// TIA Portal V19 export
FUNCTION "ALARM" : Void   // FC6, LAD
{ S7_Optimized_Access := 'TRUE' }
// stored: SetENOAutomatically false
   VAR_TEMP   // added for the SCL form of the ladder/FBD networks
      _w1 : Bool;
      _w2 : Bool;
   END_VAR
BEGIN

REGION Network 1: ALARM RESET (MASTER TO SLAVE)
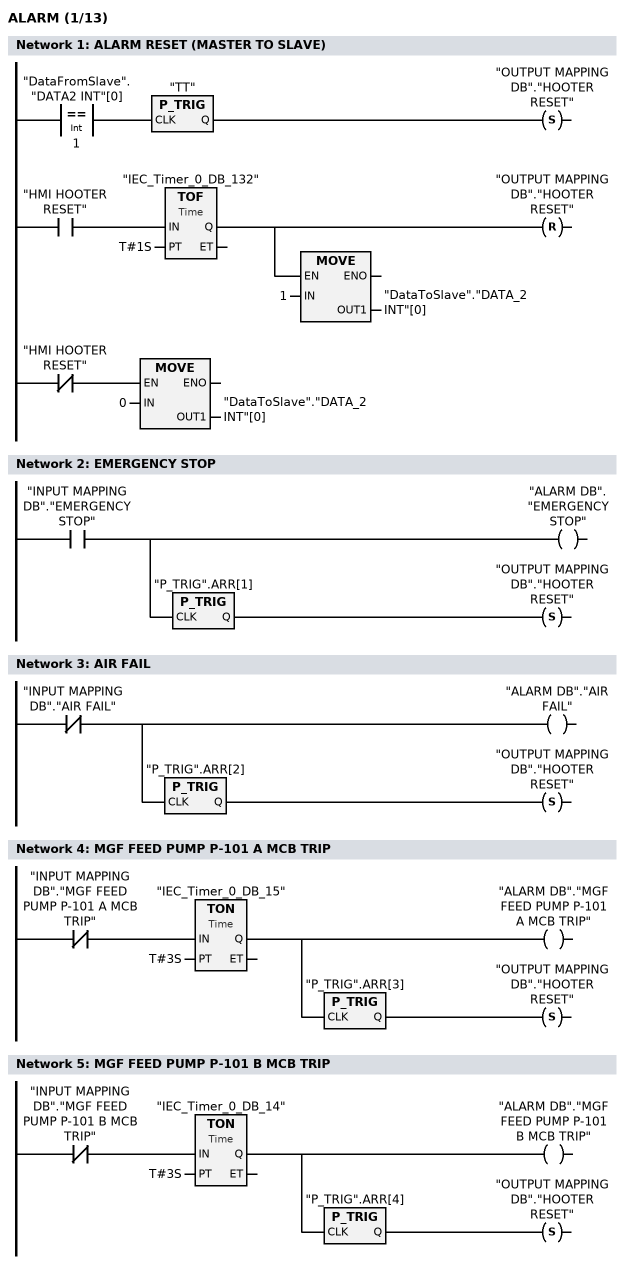
   RUNG wire#powerrail
      { S7_Templates := "SrcType := Int" } EQ_Contact(in1 := "DataFromSlave"."DATA2 INT"[0], in2 := 1)
      P_Trig( "TT" )
      S_Coil( "OUTPUT MAPPING DB"."HOOTER RESET" )
   END_RUNG
   RUNG wire#powerrail
      Contact( "HMI HOOTER RESET" )
      { S7_Templates := "time_type := Time" } "IEC_Timer_0_DB_132".TOF(pt := T#1S, et =>)
      wire#w1
      R_Coil( "OUTPUT MAPPING DB"."HOOTER RESET" )
   END_RUNG
   RUNG wire#w1
      Move(in := 1, out1 => "DataToSlave"."DATA_2 INT"[0])
   END_RUNG
   RUNG wire#powerrail
      I_Contact( "HMI HOOTER RESET" )
      Move(in := 0, out1 => "DataToSlave"."DATA_2 INT"[0])
   END_RUNG
   // the same network as SCL:
   #_w1 := "DataFromSlave"."DATA2 INT"[0] = 1;
   #_w2 := #_w1 AND NOT "TT";   // rising edge
   "TT" := #_w1;
   IF #_w2 THEN "OUTPUT MAPPING DB"."HOOTER RESET" := TRUE; END_IF;
   "IEC_Timer_0_DB_132".TOF(IN := "HMI HOOTER RESET", PT := T#1S);
   IF "IEC_Timer_0_DB_132".Q THEN
       "OUTPUT MAPPING DB"."HOOTER RESET" := FALSE;
       "DataToSlave"."DATA_2 INT"[0] := 1;
   END_IF;
   IF NOT "HMI HOOTER RESET" THEN "DataToSlave"."DATA_2 INT"[0] := 0; END_IF;
END_REGION

REGION Network 2: EMERGENCY STOP
   RUNG wire#powerrail
      Contact( "INPUT MAPPING DB"."EMERGENCY STOP" )
      wire#w1
      Coil( "ALARM DB"."EMERGENCY STOP" )
   END_RUNG
   RUNG wire#w1
      P_Trig( "P_TRIG".ARR[1] )
      S_Coil( "OUTPUT MAPPING DB"."HOOTER RESET" )
   END_RUNG
   // the same network as SCL:
   "ALARM DB"."EMERGENCY STOP" := "INPUT MAPPING DB"."EMERGENCY STOP";
   #_w1 := "INPUT MAPPING DB"."EMERGENCY STOP" AND NOT "P_TRIG".ARR[1];   // rising edge
   "P_TRIG".ARR[1] := "INPUT MAPPING DB"."EMERGENCY STOP";
   IF #_w1 THEN "OUTPUT MAPPING DB"."HOOTER RESET" := TRUE; END_IF;
END_REGION

REGION Network 3: AIR FAIL
   RUNG wire#powerrail
      I_Contact( "INPUT MAPPING DB"."AIR FAIL" )
      wire#w1
      Coil( "ALARM DB"."AIR FAIL" )
   END_RUNG
   RUNG wire#w1
      P_Trig( "P_TRIG".ARR[2] )
      S_Coil( "OUTPUT MAPPING DB"."HOOTER RESET" )
   END_RUNG
   // the same network as SCL:
   "ALARM DB"."AIR FAIL" := NOT "INPUT MAPPING DB"."AIR FAIL";
   #_w1 := NOT "INPUT MAPPING DB"."AIR FAIL" AND NOT "P_TRIG".ARR[2];   // rising edge
   "P_TRIG".ARR[2] := NOT "INPUT MAPPING DB"."AIR FAIL";
   IF #_w1 THEN "OUTPUT MAPPING DB"."HOOTER RESET" := TRUE; END_IF;
END_REGION

REGION Network 4: MGF FEED PUMP P-101 A MCB TRIP
   RUNG wire#powerrail
      I_Contact( "INPUT MAPPING DB"."MGF FEED PUMP P-101 A MCB TRIP" )
      { S7_Templates := "time_type := Time" } "IEC_Timer_0_DB_15".TON(pt := T#3S, et =>)
      wire#w1
      Coil( "ALARM DB"."MGF FEED PUMP P-101 A MCB TRIP" )
   END_RUNG
   RUNG wire#w1
      P_Trig( "P_TRIG".ARR[3] )
      S_Coil( "OUTPUT MAPPING DB"."HOOTER RESET" )
   END_RUNG
   // the same network as SCL:
   "IEC_Timer_0_DB_15".TON(IN := NOT "INPUT MAPPING DB"."MGF FEED PUMP P-101 A MCB TRIP", PT := T#3S);
   "ALARM DB"."MGF FEED PUMP P-101 A MCB TRIP" := "IEC_Timer_0_DB_15".Q;
   #_w1 := "IEC_Timer_0_DB_15".Q AND NOT "P_TRIG".ARR[3];   // rising edge
   "P_TRIG".ARR[3] := "IEC_Timer_0_DB_15".Q;
   IF #_w1 THEN "OUTPUT MAPPING DB"."HOOTER RESET" := TRUE; END_IF;
END_REGION

REGION Network 5: MGF FEED PUMP P-101 B MCB TRIP
   RUNG wire#powerrail
      I_Contact( "INPUT MAPPING DB"."MGF FEED PUMP P-101 B MCB TRIP" )
      { S7_Templates := "time_type := Time" } "IEC_Timer_0_DB_14".TON(pt := T#3S, et =>)
      wire#w1
      Coil( "ALARM DB"."MGF FEED PUMP P-101 B MCB TRIP" )
   END_RUNG
   RUNG wire#w1
      P_Trig( "P_TRIG".ARR[4] )
      S_Coil( "OUTPUT MAPPING DB"."HOOTER RESET" )
   END_RUNG
   // the same network as SCL:
   "IEC_Timer_0_DB_14".TON(IN := NOT "INPUT MAPPING DB"."MGF FEED PUMP P-101 B MCB TRIP", PT := T#3S);
   "ALARM DB"."MGF FEED PUMP P-101 B MCB TRIP" := "IEC_Timer_0_DB_14".Q;
   #_w1 := "IEC_Timer_0_DB_14".Q AND NOT "P_TRIG".ARR[4];   // rising edge
   "P_TRIG".ARR[4] := "IEC_Timer_0_DB_14".Q;
   IF #_w1 THEN "OUTPUT MAPPING DB"."HOOTER RESET" := TRUE; END_IF;
END_REGION

REGION Network 6: MGF BACK WASH P-102 A MCB TRIP
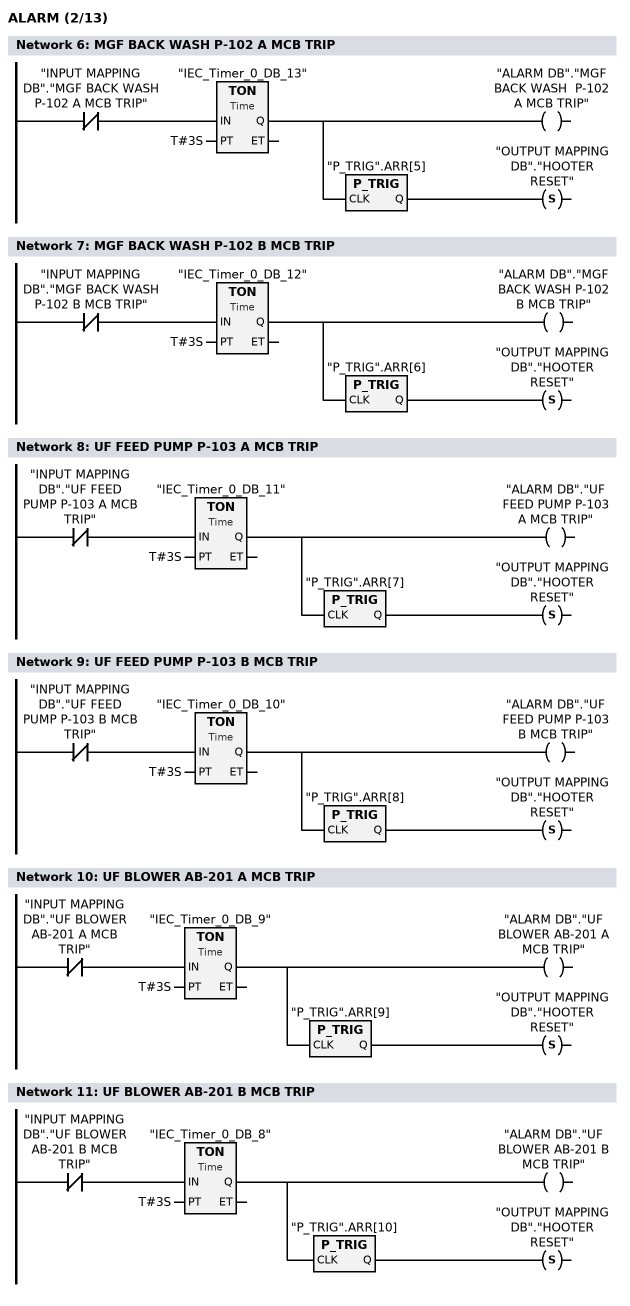
   RUNG wire#powerrail
      I_Contact( "INPUT MAPPING DB"."MGF BACK WASH  P-102 A MCB TRIP" )
      { S7_Templates := "time_type := Time" } "IEC_Timer_0_DB_13".TON(pt := T#3S, et =>)
      wire#w1
      Coil( "ALARM DB"."MGF BACK WASH  P-102 A MCB TRIP" )
   END_RUNG
   RUNG wire#w1
      P_Trig( "P_TRIG".ARR[5] )
      S_Coil( "OUTPUT MAPPING DB"."HOOTER RESET" )
   END_RUNG
   // the same network as SCL:
   "IEC_Timer_0_DB_13".TON(IN := NOT "INPUT MAPPING DB"."MGF BACK WASH  P-102 A MCB TRIP", PT := T#3S);
   "ALARM DB"."MGF BACK WASH  P-102 A MCB TRIP" := "IEC_Timer_0_DB_13".Q;
   #_w1 := "IEC_Timer_0_DB_13".Q AND NOT "P_TRIG".ARR[5];   // rising edge
   "P_TRIG".ARR[5] := "IEC_Timer_0_DB_13".Q;
   IF #_w1 THEN "OUTPUT MAPPING DB"."HOOTER RESET" := TRUE; END_IF;
END_REGION

REGION Network 7: MGF BACK WASH P-102 B MCB TRIP
   RUNG wire#powerrail
      I_Contact( "INPUT MAPPING DB"."MGF BACK WASH P-102 B MCB TRIP" )
      { S7_Templates := "time_type := Time" } "IEC_Timer_0_DB_12".TON(pt := T#3S, et =>)
      wire#w1
      Coil( "ALARM DB"."MGF BACK WASH P-102 B MCB TRIP" )
   END_RUNG
   RUNG wire#w1
      P_Trig( "P_TRIG".ARR[6] )
      S_Coil( "OUTPUT MAPPING DB"."HOOTER RESET" )
   END_RUNG
   // the same network as SCL:
   "IEC_Timer_0_DB_12".TON(IN := NOT "INPUT MAPPING DB"."MGF BACK WASH P-102 B MCB TRIP", PT := T#3S);
   "ALARM DB"."MGF BACK WASH P-102 B MCB TRIP" := "IEC_Timer_0_DB_12".Q;
   #_w1 := "IEC_Timer_0_DB_12".Q AND NOT "P_TRIG".ARR[6];   // rising edge
   "P_TRIG".ARR[6] := "IEC_Timer_0_DB_12".Q;
   IF #_w1 THEN "OUTPUT MAPPING DB"."HOOTER RESET" := TRUE; END_IF;
END_REGION

REGION Network 8: UF FEED PUMP P-103 A MCB TRIP
   RUNG wire#powerrail
      I_Contact( "INPUT MAPPING DB"."UF FEED PUMP P-103 A MCB TRIP" )
      { S7_Templates := "time_type := Time" } "IEC_Timer_0_DB_11".TON(pt := T#3S, et =>)
      wire#w1
      Coil( "ALARM DB"."UF FEED PUMP P-103 A MCB TRIP" )
   END_RUNG
   RUNG wire#w1
      P_Trig( "P_TRIG".ARR[7] )
      S_Coil( "OUTPUT MAPPING DB"."HOOTER RESET" )
   END_RUNG
   // the same network as SCL:
   "IEC_Timer_0_DB_11".TON(IN := NOT "INPUT MAPPING DB"."UF FEED PUMP P-103 A MCB TRIP", PT := T#3S);
   "ALARM DB"."UF FEED PUMP P-103 A MCB TRIP" := "IEC_Timer_0_DB_11".Q;
   #_w1 := "IEC_Timer_0_DB_11".Q AND NOT "P_TRIG".ARR[7];   // rising edge
   "P_TRIG".ARR[7] := "IEC_Timer_0_DB_11".Q;
   IF #_w1 THEN "OUTPUT MAPPING DB"."HOOTER RESET" := TRUE; END_IF;
END_REGION

REGION Network 9: UF FEED PUMP P-103 B MCB TRIP
   RUNG wire#powerrail
      I_Contact( "INPUT MAPPING DB"."UF FEED PUMP P-103 B MCB TRIP" )
      { S7_Templates := "time_type := Time" } "IEC_Timer_0_DB_10".TON(pt := T#3S, et =>)
      wire#w1
      Coil( "ALARM DB"."UF FEED PUMP P-103 B MCB TRIP" )
   END_RUNG
   RUNG wire#w1
      P_Trig( "P_TRIG".ARR[8] )
      S_Coil( "OUTPUT MAPPING DB"."HOOTER RESET" )
   END_RUNG
   // the same network as SCL:
   "IEC_Timer_0_DB_10".TON(IN := NOT "INPUT MAPPING DB"."UF FEED PUMP P-103 B MCB TRIP", PT := T#3S);
   "ALARM DB"."UF FEED PUMP P-103 B MCB TRIP" := "IEC_Timer_0_DB_10".Q;
   #_w1 := "IEC_Timer_0_DB_10".Q AND NOT "P_TRIG".ARR[8];   // rising edge
   "P_TRIG".ARR[8] := "IEC_Timer_0_DB_10".Q;
   IF #_w1 THEN "OUTPUT MAPPING DB"."HOOTER RESET" := TRUE; END_IF;
END_REGION

REGION Network 10: UF BLOWER AB-201 A MCB TRIP
   RUNG wire#powerrail
      I_Contact( "INPUT MAPPING DB"."UF BLOWER AB-201 A MCB TRIP" )
      { S7_Templates := "time_type := Time" } "IEC_Timer_0_DB_9".TON(pt := T#3S, et =>)
      wire#w1
      Coil( "ALARM DB"."UF BLOWER AB-201 A MCB TRIP" )
   END_RUNG
   RUNG wire#w1
      P_Trig( "P_TRIG".ARR[9] )
      S_Coil( "OUTPUT MAPPING DB"."HOOTER RESET" )
   END_RUNG
   // the same network as SCL:
   "IEC_Timer_0_DB_9".TON(IN := NOT "INPUT MAPPING DB"."UF BLOWER AB-201 A MCB TRIP", PT := T#3S);
   "ALARM DB"."UF BLOWER AB-201 A MCB TRIP" := "IEC_Timer_0_DB_9".Q;
   #_w1 := "IEC_Timer_0_DB_9".Q AND NOT "P_TRIG".ARR[9];   // rising edge
   "P_TRIG".ARR[9] := "IEC_Timer_0_DB_9".Q;
   IF #_w1 THEN "OUTPUT MAPPING DB"."HOOTER RESET" := TRUE; END_IF;
END_REGION

REGION Network 11: UF BLOWER AB-201 B MCB TRIP
   RUNG wire#powerrail
      I_Contact( "INPUT MAPPING DB"."UF BLOWER AB-201 B MCB TRIP" )
      { S7_Templates := "time_type := Time" } "IEC_Timer_0_DB_8".TON(pt := T#3S, et =>)
      wire#w1
      Coil( "ALARM DB"."UF BLOWER AB-201 B MCB TRIP" )
   END_RUNG
   RUNG wire#w1
      P_Trig( "P_TRIG".ARR[10] )
      S_Coil( "OUTPUT MAPPING DB"."HOOTER RESET" )
   END_RUNG
   // the same network as SCL:
   "IEC_Timer_0_DB_8".TON(IN := NOT "INPUT MAPPING DB"."UF BLOWER AB-201 B MCB TRIP", PT := T#3S);
   "ALARM DB"."UF BLOWER AB-201 B MCB TRIP" := "IEC_Timer_0_DB_8".Q;
   #_w1 := "IEC_Timer_0_DB_8".Q AND NOT "P_TRIG".ARR[10];   // rising edge
   "P_TRIG".ARR[10] := "IEC_Timer_0_DB_8".Q;
   IF #_w1 THEN "OUTPUT MAPPING DB"."HOOTER RESET" := TRUE; END_IF;
END_REGION

REGION Network 12: DM FEED PUMP P-502 A MPCB TRIP
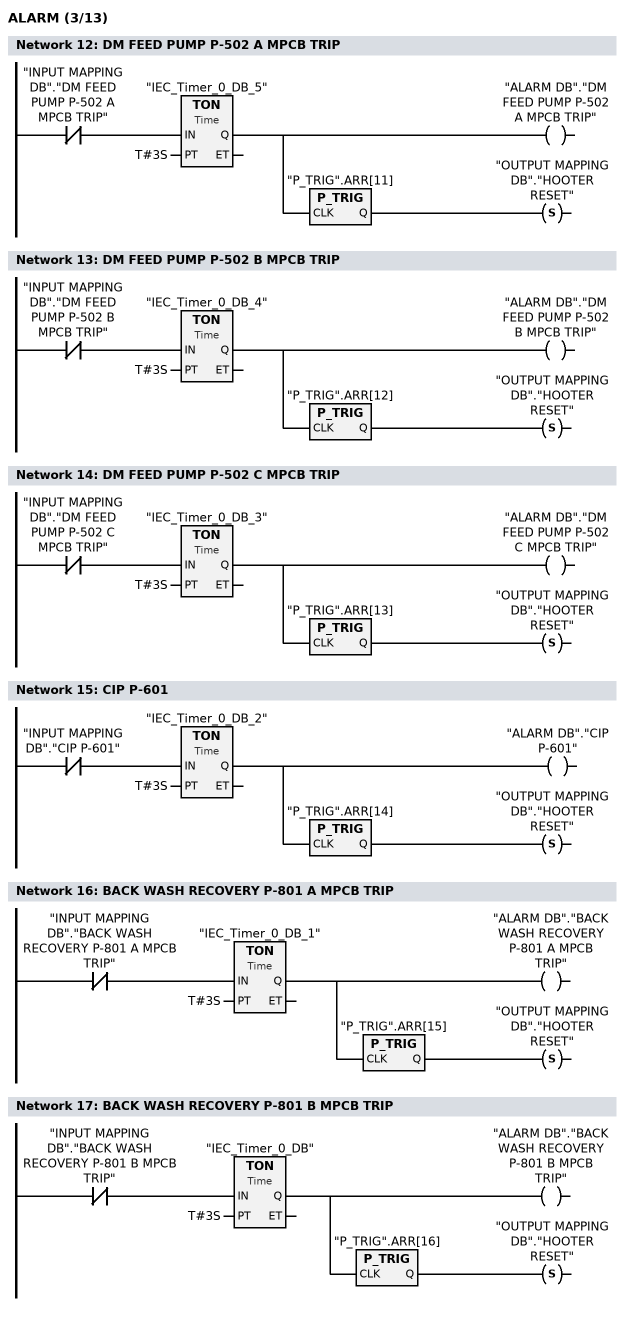
   RUNG wire#powerrail
      I_Contact( "INPUT MAPPING DB"."DM FEED PUMP P-502 A MPCB TRIP" )
      { S7_Templates := "time_type := Time" } "IEC_Timer_0_DB_5".TON(pt := T#3S, et =>)
      wire#w1
      Coil( "ALARM DB"."DM FEED PUMP P-502 A MPCB TRIP" )
   END_RUNG
   RUNG wire#w1
      P_Trig( "P_TRIG".ARR[11] )
      S_Coil( "OUTPUT MAPPING DB"."HOOTER RESET" )
   END_RUNG
   // the same network as SCL:
   "IEC_Timer_0_DB_5".TON(IN := NOT "INPUT MAPPING DB"."DM FEED PUMP P-502 A MPCB TRIP", PT := T#3S);
   "ALARM DB"."DM FEED PUMP P-502 A MPCB TRIP" := "IEC_Timer_0_DB_5".Q;
   #_w1 := "IEC_Timer_0_DB_5".Q AND NOT "P_TRIG".ARR[11];   // rising edge
   "P_TRIG".ARR[11] := "IEC_Timer_0_DB_5".Q;
   IF #_w1 THEN "OUTPUT MAPPING DB"."HOOTER RESET" := TRUE; END_IF;
END_REGION

REGION Network 13: DM FEED PUMP P-502 B MPCB TRIP
   RUNG wire#powerrail
      I_Contact( "INPUT MAPPING DB"."DM FEED PUMP P-502 B MPCB TRIP" )
      { S7_Templates := "time_type := Time" } "IEC_Timer_0_DB_4".TON(pt := T#3S, et =>)
      wire#w1
      Coil( "ALARM DB"."DM FEED PUMP P-502 B MPCB TRIP" )
   END_RUNG
   RUNG wire#w1
      P_Trig( "P_TRIG".ARR[12] )
      S_Coil( "OUTPUT MAPPING DB"."HOOTER RESET" )
   END_RUNG
   // the same network as SCL:
   "IEC_Timer_0_DB_4".TON(IN := NOT "INPUT MAPPING DB"."DM FEED PUMP P-502 B MPCB TRIP", PT := T#3S);
   "ALARM DB"."DM FEED PUMP P-502 B MPCB TRIP" := "IEC_Timer_0_DB_4".Q;
   #_w1 := "IEC_Timer_0_DB_4".Q AND NOT "P_TRIG".ARR[12];   // rising edge
   "P_TRIG".ARR[12] := "IEC_Timer_0_DB_4".Q;
   IF #_w1 THEN "OUTPUT MAPPING DB"."HOOTER RESET" := TRUE; END_IF;
END_REGION

REGION Network 14: DM FEED PUMP P-502 C MPCB TRIP
   RUNG wire#powerrail
      I_Contact( "INPUT MAPPING DB"."DM FEED PUMP P-502 C MPCB TRIP" )
      { S7_Templates := "time_type := Time" } "IEC_Timer_0_DB_3".TON(pt := T#3S, et =>)
      wire#w1
      Coil( "ALARM DB"."DM FEED PUMP P-502 C MPCB TRIP" )
   END_RUNG
   RUNG wire#w1
      P_Trig( "P_TRIG".ARR[13] )
      S_Coil( "OUTPUT MAPPING DB"."HOOTER RESET" )
   END_RUNG
   // the same network as SCL:
   "IEC_Timer_0_DB_3".TON(IN := NOT "INPUT MAPPING DB"."DM FEED PUMP P-502 C MPCB TRIP", PT := T#3S);
   "ALARM DB"."DM FEED PUMP P-502 C MPCB TRIP" := "IEC_Timer_0_DB_3".Q;
   #_w1 := "IEC_Timer_0_DB_3".Q AND NOT "P_TRIG".ARR[13];   // rising edge
   "P_TRIG".ARR[13] := "IEC_Timer_0_DB_3".Q;
   IF #_w1 THEN "OUTPUT MAPPING DB"."HOOTER RESET" := TRUE; END_IF;
END_REGION

REGION Network 15: CIP P-601
   RUNG wire#powerrail
      I_Contact( "INPUT MAPPING DB"."CIP P-601" )
      { S7_Templates := "time_type := Time" } "IEC_Timer_0_DB_2".TON(pt := T#3S, et =>)
      wire#w1
      Coil( "ALARM DB"."CIP P-601" )
   END_RUNG
   RUNG wire#w1
      P_Trig( "P_TRIG".ARR[14] )
      S_Coil( "OUTPUT MAPPING DB"."HOOTER RESET" )
   END_RUNG
   // the same network as SCL:
   "IEC_Timer_0_DB_2".TON(IN := NOT "INPUT MAPPING DB"."CIP P-601", PT := T#3S);
   "ALARM DB"."CIP P-601" := "IEC_Timer_0_DB_2".Q;
   #_w1 := "IEC_Timer_0_DB_2".Q AND NOT "P_TRIG".ARR[14];   // rising edge
   "P_TRIG".ARR[14] := "IEC_Timer_0_DB_2".Q;
   IF #_w1 THEN "OUTPUT MAPPING DB"."HOOTER RESET" := TRUE; END_IF;
END_REGION

REGION Network 16: BACK WASH RECOVERY P-801 A MPCB TRIP
   RUNG wire#powerrail
      I_Contact( "INPUT MAPPING DB"."BACK WASH RECOVERY P-801 A MPCB TRIP" )
      { S7_Templates := "time_type := Time" } "IEC_Timer_0_DB_1".TON(pt := T#3S, et =>)
      wire#w1
      Coil( "ALARM DB"."BACK WASH RECOVERY P-801 A MPCB TRIP" )
   END_RUNG
   RUNG wire#w1
      P_Trig( "P_TRIG".ARR[15] )
      S_Coil( "OUTPUT MAPPING DB"."HOOTER RESET" )
   END_RUNG
   // the same network as SCL:
   "IEC_Timer_0_DB_1".TON(IN := NOT "INPUT MAPPING DB"."BACK WASH RECOVERY P-801 A MPCB TRIP", PT := T#3S);
   "ALARM DB"."BACK WASH RECOVERY P-801 A MPCB TRIP" := "IEC_Timer_0_DB_1".Q;
   #_w1 := "IEC_Timer_0_DB_1".Q AND NOT "P_TRIG".ARR[15];   // rising edge
   "P_TRIG".ARR[15] := "IEC_Timer_0_DB_1".Q;
   IF #_w1 THEN "OUTPUT MAPPING DB"."HOOTER RESET" := TRUE; END_IF;
END_REGION

REGION Network 17: BACK WASH RECOVERY P-801 B MPCB TRIP
   RUNG wire#powerrail
      I_Contact( "INPUT MAPPING DB"."BACK WASH RECOVERY P-801 B MPCB TRIP" )
      { S7_Templates := "time_type := Time" } "IEC_Timer_0_DB".TON(pt := T#3S, et =>)
      wire#w1
      Coil( "ALARM DB"."BACK WASH RECOVERY P-801 B MPCB TRIP" )
   END_RUNG
   RUNG wire#w1
      P_Trig( "P_TRIG".ARR[16] )
      S_Coil( "OUTPUT MAPPING DB"."HOOTER RESET" )
   END_RUNG
   // the same network as SCL:
   "IEC_Timer_0_DB".TON(IN := NOT "INPUT MAPPING DB"."BACK WASH RECOVERY P-801 B MPCB TRIP", PT := T#3S);
   "ALARM DB"."BACK WASH RECOVERY P-801 B MPCB TRIP" := "IEC_Timer_0_DB".Q;
   #_w1 := "IEC_Timer_0_DB".Q AND NOT "P_TRIG".ARR[16];   // rising edge
   "P_TRIG".ARR[16] := "IEC_Timer_0_DB".Q;
   IF #_w1 THEN "OUTPUT MAPPING DB"."HOOTER RESET" := TRUE; END_IF;
END_REGION

REGION Network 18: UF BACKWASH P-201A TRIP
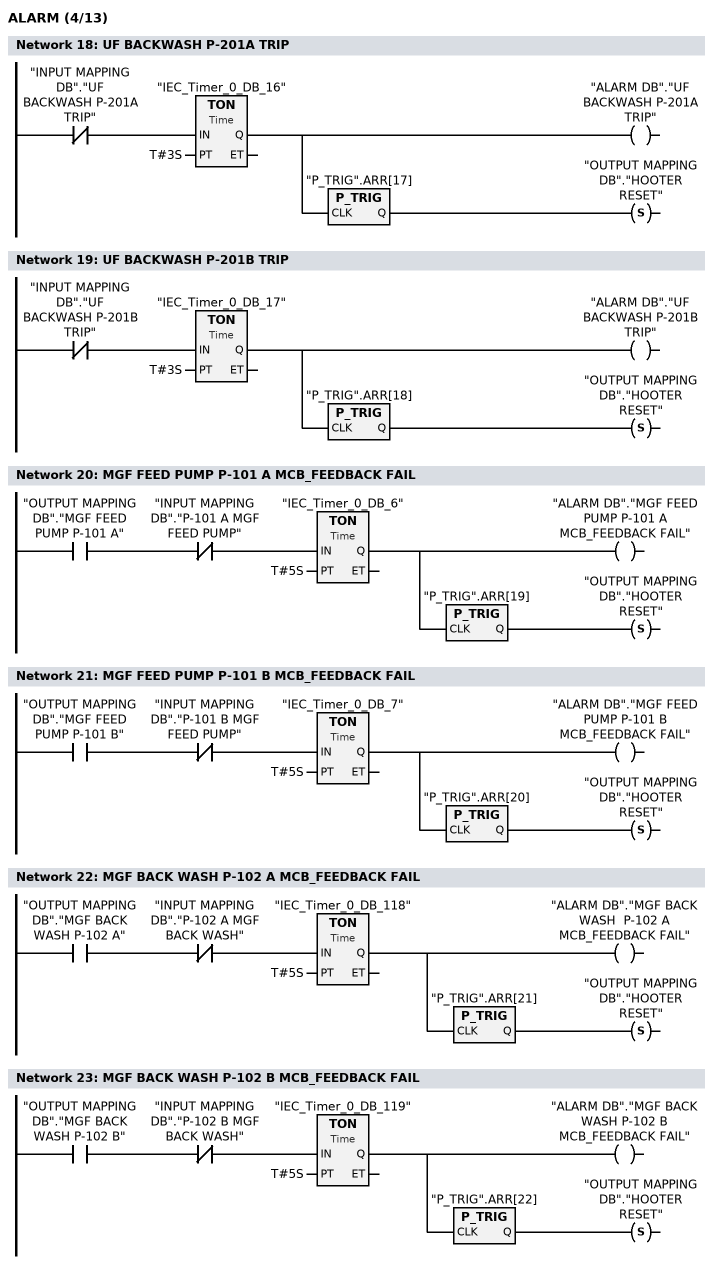
   RUNG wire#powerrail
      I_Contact( "INPUT MAPPING DB"."UF BACKWASH P-201A TRIP" )
      { S7_Templates := "time_type := Time" } "IEC_Timer_0_DB_16".TON(pt := T#3S, et =>)
      wire#w1
      Coil( "ALARM DB"."UF BACKWASH P-201A TRIP" )
   END_RUNG
   RUNG wire#w1
      P_Trig( "P_TRIG".ARR[17] )
      S_Coil( "OUTPUT MAPPING DB"."HOOTER RESET" )
   END_RUNG
   // the same network as SCL:
   "IEC_Timer_0_DB_16".TON(IN := NOT "INPUT MAPPING DB"."UF BACKWASH P-201A TRIP", PT := T#3S);
   "ALARM DB"."UF BACKWASH P-201A TRIP" := "IEC_Timer_0_DB_16".Q;
   #_w1 := "IEC_Timer_0_DB_16".Q AND NOT "P_TRIG".ARR[17];   // rising edge
   "P_TRIG".ARR[17] := "IEC_Timer_0_DB_16".Q;
   IF #_w1 THEN "OUTPUT MAPPING DB"."HOOTER RESET" := TRUE; END_IF;
END_REGION

REGION Network 19: UF BACKWASH P-201B TRIP
   RUNG wire#powerrail
      I_Contact( "INPUT MAPPING DB"."UF BACKWASH P-201B TRIP" )
      { S7_Templates := "time_type := Time" } "IEC_Timer_0_DB_17".TON(pt := T#3S, et =>)
      wire#w1
      Coil( "ALARM DB"."UF BACKWASH P-201B TRIP" )
   END_RUNG
   RUNG wire#w1
      P_Trig( "P_TRIG".ARR[18] )
      S_Coil( "OUTPUT MAPPING DB"."HOOTER RESET" )
   END_RUNG
   // the same network as SCL:
   "IEC_Timer_0_DB_17".TON(IN := NOT "INPUT MAPPING DB"."UF BACKWASH P-201B TRIP", PT := T#3S);
   "ALARM DB"."UF BACKWASH P-201B TRIP" := "IEC_Timer_0_DB_17".Q;
   #_w1 := "IEC_Timer_0_DB_17".Q AND NOT "P_TRIG".ARR[18];   // rising edge
   "P_TRIG".ARR[18] := "IEC_Timer_0_DB_17".Q;
   IF #_w1 THEN "OUTPUT MAPPING DB"."HOOTER RESET" := TRUE; END_IF;
END_REGION

REGION Network 20: MGF FEED PUMP P-101 A MCB_FEEDBACK FAIL
   RUNG wire#powerrail
      Contact( "OUTPUT MAPPING DB"."MGF FEED PUMP P-101 A" )
      I_Contact( "INPUT MAPPING DB"."P-101 A MGF FEED PUMP" )
      { S7_Templates := "time_type := Time" } "IEC_Timer_0_DB_6".TON(pt := T#5S, et =>)
      wire#w1
      Coil( "ALARM DB"."MGF FEED PUMP P-101 A MCB_FEEDBACK FAIL" )
   END_RUNG
   RUNG wire#w1
      P_Trig( "P_TRIG".ARR[19] )
      S_Coil( "OUTPUT MAPPING DB"."HOOTER RESET" )
   END_RUNG
   // the same network as SCL:
   "IEC_Timer_0_DB_6".TON(IN := "OUTPUT MAPPING DB"."MGF FEED PUMP P-101 A" AND NOT "INPUT MAPPING DB"."P-101 A MGF FEED PUMP",
                          PT := T#5S);
   "ALARM DB"."MGF FEED PUMP P-101 A MCB_FEEDBACK FAIL" := "IEC_Timer_0_DB_6".Q;
   #_w1 := "IEC_Timer_0_DB_6".Q AND NOT "P_TRIG".ARR[19];   // rising edge
   "P_TRIG".ARR[19] := "IEC_Timer_0_DB_6".Q;
   IF #_w1 THEN "OUTPUT MAPPING DB"."HOOTER RESET" := TRUE; END_IF;
END_REGION

REGION Network 21: MGF FEED PUMP P-101 B MCB_FEEDBACK FAIL
   RUNG wire#powerrail
      Contact( "OUTPUT MAPPING DB"."MGF FEED PUMP P-101 B" )
      I_Contact( "INPUT MAPPING DB"."P-101 B MGF FEED PUMP" )
      { S7_Templates := "time_type := Time" } "IEC_Timer_0_DB_7".TON(pt := T#5S, et =>)
      wire#w1
      Coil( "ALARM DB"."MGF FEED PUMP P-101 B MCB_FEEDBACK FAIL" )
   END_RUNG
   RUNG wire#w1
      P_Trig( "P_TRIG".ARR[20] )
      S_Coil( "OUTPUT MAPPING DB"."HOOTER RESET" )
   END_RUNG
   // the same network as SCL:
   "IEC_Timer_0_DB_7".TON(IN := "OUTPUT MAPPING DB"."MGF FEED PUMP P-101 B" AND NOT "INPUT MAPPING DB"."P-101 B MGF FEED PUMP",
                          PT := T#5S);
   "ALARM DB"."MGF FEED PUMP P-101 B MCB_FEEDBACK FAIL" := "IEC_Timer_0_DB_7".Q;
   #_w1 := "IEC_Timer_0_DB_7".Q AND NOT "P_TRIG".ARR[20];   // rising edge
   "P_TRIG".ARR[20] := "IEC_Timer_0_DB_7".Q;
   IF #_w1 THEN "OUTPUT MAPPING DB"."HOOTER RESET" := TRUE; END_IF;
END_REGION

REGION Network 22: MGF BACK WASH P-102 A MCB_FEEDBACK FAIL
   RUNG wire#powerrail
      Contact( "OUTPUT MAPPING DB"."MGF BACK WASH P-102 A" )
      I_Contact( "INPUT MAPPING DB"."P-102 A MGF BACK WASH" )
      { S7_Templates := "time_type := Time" } "IEC_Timer_0_DB_118".TON(pt := T#5S, et =>)
      wire#w1
      Coil( "ALARM DB"."MGF BACK WASH  P-102 A MCB_FEEDBACK FAIL" )
   END_RUNG
   RUNG wire#w1
      P_Trig( "P_TRIG".ARR[21] )
      S_Coil( "OUTPUT MAPPING DB"."HOOTER RESET" )
   END_RUNG
   // the same network as SCL:
   "IEC_Timer_0_DB_118".TON(IN := "OUTPUT MAPPING DB"."MGF BACK WASH P-102 A" AND NOT "INPUT MAPPING DB"."P-102 A MGF BACK WASH",
                           PT := T#5S);
   "ALARM DB"."MGF BACK WASH  P-102 A MCB_FEEDBACK FAIL" := "IEC_Timer_0_DB_118".Q;
   #_w1 := "IEC_Timer_0_DB_118".Q AND NOT "P_TRIG".ARR[21];   // rising edge
   "P_TRIG".ARR[21] := "IEC_Timer_0_DB_118".Q;
   IF #_w1 THEN "OUTPUT MAPPING DB"."HOOTER RESET" := TRUE; END_IF;
END_REGION

REGION Network 23: MGF BACK WASH P-102 B MCB_FEEDBACK FAIL
   RUNG wire#powerrail
      Contact( "OUTPUT MAPPING DB"."MGF BACK WASH P-102 B" )
      I_Contact( "INPUT MAPPING DB"."P-102 B MGF BACK WASH" )
      { S7_Templates := "time_type := Time" } "IEC_Timer_0_DB_119".TON(pt := T#5S, et =>)
      wire#w1
      Coil( "ALARM DB"."MGF BACK WASH P-102 B MCB_FEEDBACK FAIL" )
   END_RUNG
   RUNG wire#w1
      P_Trig( "P_TRIG".ARR[22] )
      S_Coil( "OUTPUT MAPPING DB"."HOOTER RESET" )
   END_RUNG
   // the same network as SCL:
   "IEC_Timer_0_DB_119".TON(IN := "OUTPUT MAPPING DB"."MGF BACK WASH P-102 B" AND NOT "INPUT MAPPING DB"."P-102 B MGF BACK WASH",
                           PT := T#5S);
   "ALARM DB"."MGF BACK WASH P-102 B MCB_FEEDBACK FAIL" := "IEC_Timer_0_DB_119".Q;
   #_w1 := "IEC_Timer_0_DB_119".Q AND NOT "P_TRIG".ARR[22];   // rising edge
   "P_TRIG".ARR[22] := "IEC_Timer_0_DB_119".Q;
   IF #_w1 THEN "OUTPUT MAPPING DB"."HOOTER RESET" := TRUE; END_IF;
END_REGION

REGION Network 24: UF FEED PUMP P-103 A MCB_FEEDBACK FAIL
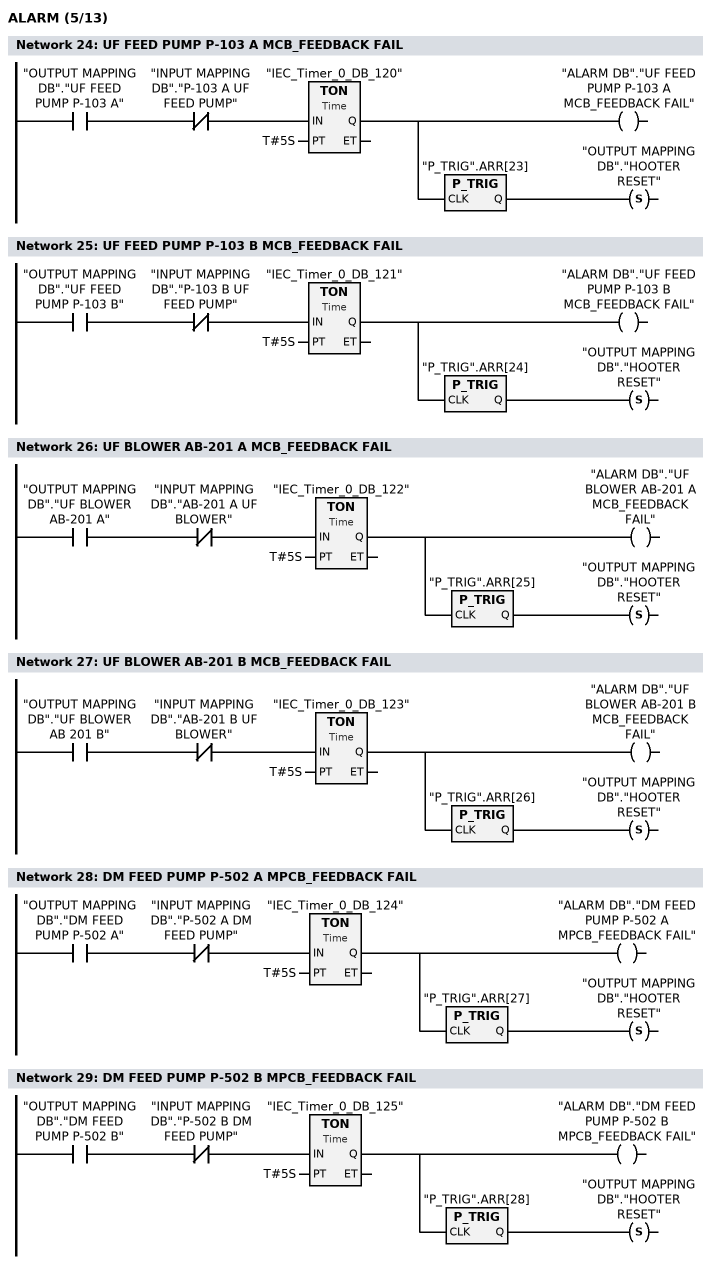
   RUNG wire#powerrail
      Contact( "OUTPUT MAPPING DB"."UF FEED PUMP P-103 A" )
      I_Contact( "INPUT MAPPING DB"."P-103 A UF FEED PUMP" )
      { S7_Templates := "time_type := Time" } "IEC_Timer_0_DB_120".TON(pt := T#5S, et =>)
      wire#w1
      Coil( "ALARM DB"."UF FEED PUMP P-103 A MCB_FEEDBACK FAIL" )
   END_RUNG
   RUNG wire#w1
      P_Trig( "P_TRIG".ARR[23] )
      S_Coil( "OUTPUT MAPPING DB"."HOOTER RESET" )
   END_RUNG
   // the same network as SCL:
   "IEC_Timer_0_DB_120".TON(IN := "OUTPUT MAPPING DB"."UF FEED PUMP P-103 A" AND NOT "INPUT MAPPING DB"."P-103 A UF FEED PUMP",
                           PT := T#5S);
   "ALARM DB"."UF FEED PUMP P-103 A MCB_FEEDBACK FAIL" := "IEC_Timer_0_DB_120".Q;
   #_w1 := "IEC_Timer_0_DB_120".Q AND NOT "P_TRIG".ARR[23];   // rising edge
   "P_TRIG".ARR[23] := "IEC_Timer_0_DB_120".Q;
   IF #_w1 THEN "OUTPUT MAPPING DB"."HOOTER RESET" := TRUE; END_IF;
END_REGION

REGION Network 25: UF FEED PUMP P-103 B MCB_FEEDBACK FAIL
   RUNG wire#powerrail
      Contact( "OUTPUT MAPPING DB"."UF FEED PUMP P-103 B" )
      I_Contact( "INPUT MAPPING DB"."P-103 B UF FEED PUMP" )
      { S7_Templates := "time_type := Time" } "IEC_Timer_0_DB_121".TON(pt := T#5S, et =>)
      wire#w1
      Coil( "ALARM DB"."UF FEED PUMP P-103 B MCB_FEEDBACK FAIL" )
   END_RUNG
   RUNG wire#w1
      P_Trig( "P_TRIG".ARR[24] )
      S_Coil( "OUTPUT MAPPING DB"."HOOTER RESET" )
   END_RUNG
   // the same network as SCL:
   "IEC_Timer_0_DB_121".TON(IN := "OUTPUT MAPPING DB"."UF FEED PUMP P-103 B" AND NOT "INPUT MAPPING DB"."P-103 B UF FEED PUMP",
                           PT := T#5S);
   "ALARM DB"."UF FEED PUMP P-103 B MCB_FEEDBACK FAIL" := "IEC_Timer_0_DB_121".Q;
   #_w1 := "IEC_Timer_0_DB_121".Q AND NOT "P_TRIG".ARR[24];   // rising edge
   "P_TRIG".ARR[24] := "IEC_Timer_0_DB_121".Q;
   IF #_w1 THEN "OUTPUT MAPPING DB"."HOOTER RESET" := TRUE; END_IF;
END_REGION

REGION Network 26: UF BLOWER AB-201 A MCB_FEEDBACK FAIL
   RUNG wire#powerrail
      Contact( "OUTPUT MAPPING DB"."UF BLOWER AB-201 A" )
      I_Contact( "INPUT MAPPING DB"."AB-201 A UF BLOWER" )
      { S7_Templates := "time_type := Time" } "IEC_Timer_0_DB_122".TON(pt := T#5S, et =>)
      wire#w1
      Coil( "ALARM DB"."UF BLOWER AB-201 A MCB_FEEDBACK FAIL" )
   END_RUNG
   RUNG wire#w1
      P_Trig( "P_TRIG".ARR[25] )
      S_Coil( "OUTPUT MAPPING DB"."HOOTER RESET" )
   END_RUNG
   // the same network as SCL:
   "IEC_Timer_0_DB_122".TON(IN := "OUTPUT MAPPING DB"."UF BLOWER AB-201 A" AND NOT "INPUT MAPPING DB"."AB-201 A UF BLOWER",
                           PT := T#5S);
   "ALARM DB"."UF BLOWER AB-201 A MCB_FEEDBACK FAIL" := "IEC_Timer_0_DB_122".Q;
   #_w1 := "IEC_Timer_0_DB_122".Q AND NOT "P_TRIG".ARR[25];   // rising edge
   "P_TRIG".ARR[25] := "IEC_Timer_0_DB_122".Q;
   IF #_w1 THEN "OUTPUT MAPPING DB"."HOOTER RESET" := TRUE; END_IF;
END_REGION

REGION Network 27: UF BLOWER AB-201 B MCB_FEEDBACK FAIL
   RUNG wire#powerrail
      Contact( "OUTPUT MAPPING DB"."UF BLOWER AB 201 B" )
      I_Contact( "INPUT MAPPING DB"."AB-201 B UF BLOWER" )
      { S7_Templates := "time_type := Time" } "IEC_Timer_0_DB_123".TON(pt := T#5S, et =>)
      wire#w1
      Coil( "ALARM DB"."UF BLOWER AB-201 B MCB_FEEDBACK FAIL" )
   END_RUNG
   RUNG wire#w1
      P_Trig( "P_TRIG".ARR[26] )
      S_Coil( "OUTPUT MAPPING DB"."HOOTER RESET" )
   END_RUNG
   // the same network as SCL:
   "IEC_Timer_0_DB_123".TON(IN := "OUTPUT MAPPING DB"."UF BLOWER AB 201 B" AND NOT "INPUT MAPPING DB"."AB-201 B UF BLOWER",
                           PT := T#5S);
   "ALARM DB"."UF BLOWER AB-201 B MCB_FEEDBACK FAIL" := "IEC_Timer_0_DB_123".Q;
   #_w1 := "IEC_Timer_0_DB_123".Q AND NOT "P_TRIG".ARR[26];   // rising edge
   "P_TRIG".ARR[26] := "IEC_Timer_0_DB_123".Q;
   IF #_w1 THEN "OUTPUT MAPPING DB"."HOOTER RESET" := TRUE; END_IF;
END_REGION

REGION Network 28: DM FEED PUMP P-502 A MPCB_FEEDBACK FAIL
   RUNG wire#powerrail
      Contact( "OUTPUT MAPPING DB"."DM FEED PUMP P-502 A" )
      I_Contact( "INPUT MAPPING DB"."P-502 A DM FEED PUMP" )
      { S7_Templates := "time_type := Time" } "IEC_Timer_0_DB_124".TON(pt := T#5S, et =>)
      wire#w1
      Coil( "ALARM DB"."DM FEED PUMP P-502 A MPCB_FEEDBACK FAIL" )
   END_RUNG
   RUNG wire#w1
      P_Trig( "P_TRIG".ARR[27] )
      S_Coil( "OUTPUT MAPPING DB"."HOOTER RESET" )
   END_RUNG
   // the same network as SCL:
   "IEC_Timer_0_DB_124".TON(IN := "OUTPUT MAPPING DB"."DM FEED PUMP P-502 A" AND NOT "INPUT MAPPING DB"."P-502 A DM FEED PUMP",
                           PT := T#5S);
   "ALARM DB"."DM FEED PUMP P-502 A MPCB_FEEDBACK FAIL" := "IEC_Timer_0_DB_124".Q;
   #_w1 := "IEC_Timer_0_DB_124".Q AND NOT "P_TRIG".ARR[27];   // rising edge
   "P_TRIG".ARR[27] := "IEC_Timer_0_DB_124".Q;
   IF #_w1 THEN "OUTPUT MAPPING DB"."HOOTER RESET" := TRUE; END_IF;
END_REGION

REGION Network 29: DM FEED PUMP P-502 B MPCB_FEEDBACK FAIL
   RUNG wire#powerrail
      Contact( "OUTPUT MAPPING DB"."DM FEED PUMP P-502 B" )
      I_Contact( "INPUT MAPPING DB"."P-502 B DM FEED PUMP" )
      { S7_Templates := "time_type := Time" } "IEC_Timer_0_DB_125".TON(pt := T#5S, et =>)
      wire#w1
      Coil( "ALARM DB"."DM FEED PUMP P-502 B MPCB_FEEDBACK FAIL" )
   END_RUNG
   RUNG wire#w1
      P_Trig( "P_TRIG".ARR[28] )
      S_Coil( "OUTPUT MAPPING DB"."HOOTER RESET" )
   END_RUNG
   // the same network as SCL:
   "IEC_Timer_0_DB_125".TON(IN := "OUTPUT MAPPING DB"."DM FEED PUMP P-502 B" AND NOT "INPUT MAPPING DB"."P-502 B DM FEED PUMP",
                           PT := T#5S);
   "ALARM DB"."DM FEED PUMP P-502 B MPCB_FEEDBACK FAIL" := "IEC_Timer_0_DB_125".Q;
   #_w1 := "IEC_Timer_0_DB_125".Q AND NOT "P_TRIG".ARR[28];   // rising edge
   "P_TRIG".ARR[28] := "IEC_Timer_0_DB_125".Q;
   IF #_w1 THEN "OUTPUT MAPPING DB"."HOOTER RESET" := TRUE; END_IF;
END_REGION

REGION Network 30: DM FEED PUMP P-502 C MPCB_FEEDBACK FAIL
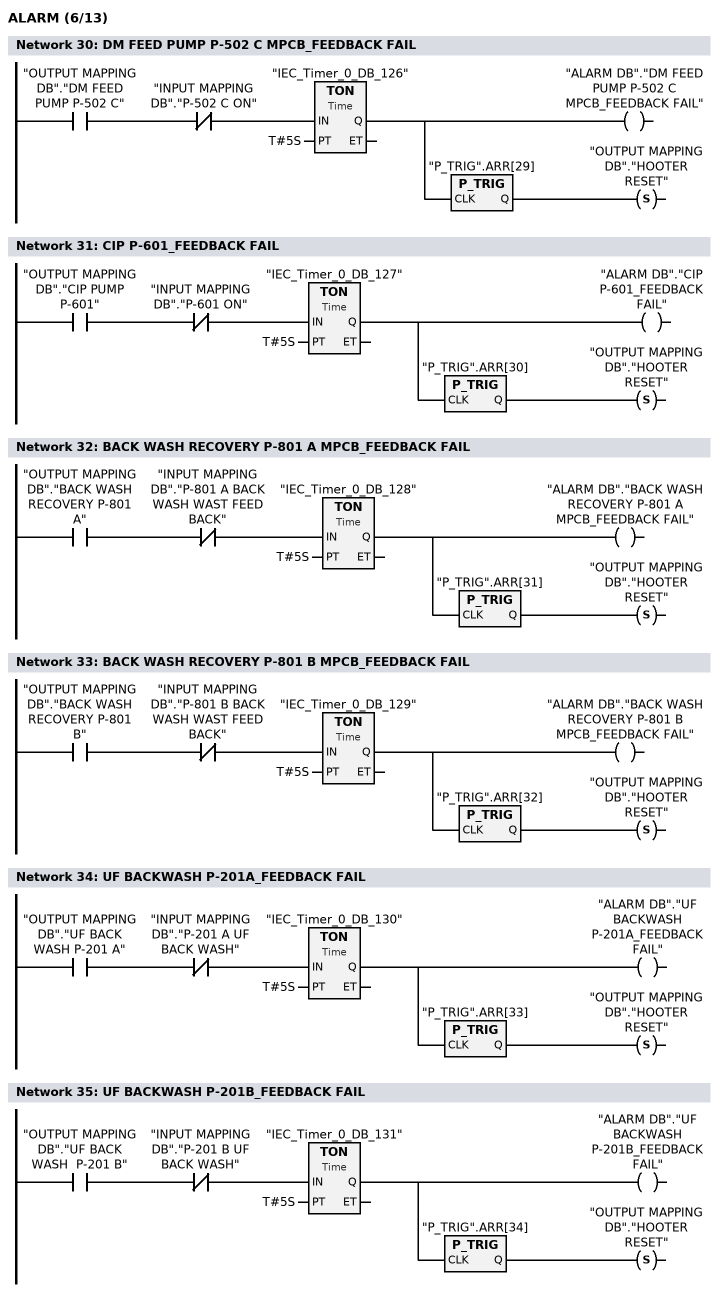
   RUNG wire#powerrail
      Contact( "OUTPUT MAPPING DB"."DM FEED PUMP P-502 C" )
      I_Contact( "INPUT MAPPING DB"."P-502 C ON" )
      { S7_Templates := "time_type := Time" } "IEC_Timer_0_DB_126".TON(pt := T#5S, et =>)
      wire#w1
      Coil( "ALARM DB"."DM FEED PUMP P-502 C MPCB_FEEDBACK FAIL" )
   END_RUNG
   RUNG wire#w1
      P_Trig( "P_TRIG".ARR[29] )
      S_Coil( "OUTPUT MAPPING DB"."HOOTER RESET" )
   END_RUNG
   // the same network as SCL:
   "IEC_Timer_0_DB_126".TON(IN := "OUTPUT MAPPING DB"."DM FEED PUMP P-502 C" AND NOT "INPUT MAPPING DB"."P-502 C ON",
                           PT := T#5S);
   "ALARM DB"."DM FEED PUMP P-502 C MPCB_FEEDBACK FAIL" := "IEC_Timer_0_DB_126".Q;
   #_w1 := "IEC_Timer_0_DB_126".Q AND NOT "P_TRIG".ARR[29];   // rising edge
   "P_TRIG".ARR[29] := "IEC_Timer_0_DB_126".Q;
   IF #_w1 THEN "OUTPUT MAPPING DB"."HOOTER RESET" := TRUE; END_IF;
END_REGION

REGION Network 31: CIP P-601_FEEDBACK FAIL
   RUNG wire#powerrail
      Contact( "OUTPUT MAPPING DB"."CIP PUMP P-601" )
      I_Contact( "INPUT MAPPING DB"."P-601 ON" )
      { S7_Templates := "time_type := Time" } "IEC_Timer_0_DB_127".TON(pt := T#5S, et =>)
      wire#w1
      Coil( "ALARM DB"."CIP P-601_FEEDBACK FAIL" )
   END_RUNG
   RUNG wire#w1
      P_Trig( "P_TRIG".ARR[30] )
      S_Coil( "OUTPUT MAPPING DB"."HOOTER RESET" )
   END_RUNG
   // the same network as SCL:
   "IEC_Timer_0_DB_127".TON(IN := "OUTPUT MAPPING DB"."CIP PUMP P-601" AND NOT "INPUT MAPPING DB"."P-601 ON",
                           PT := T#5S);
   "ALARM DB"."CIP P-601_FEEDBACK FAIL" := "IEC_Timer_0_DB_127".Q;
   #_w1 := "IEC_Timer_0_DB_127".Q AND NOT "P_TRIG".ARR[30];   // rising edge
   "P_TRIG".ARR[30] := "IEC_Timer_0_DB_127".Q;
   IF #_w1 THEN "OUTPUT MAPPING DB"."HOOTER RESET" := TRUE; END_IF;
END_REGION

REGION Network 32: BACK WASH RECOVERY P-801 A MPCB_FEEDBACK FAIL
   RUNG wire#powerrail
      Contact( "OUTPUT MAPPING DB"."BACK WASH RECOVERY P-801 A" )
      I_Contact( "INPUT MAPPING DB"."P-801 A BACK WASH WAST FEED BACK" )
      { S7_Templates := "time_type := Time" } "IEC_Timer_0_DB_128".TON(pt := T#5S, et =>)
      wire#w1
      Coil( "ALARM DB"."BACK WASH RECOVERY P-801 A MPCB_FEEDBACK FAIL" )
   END_RUNG
   RUNG wire#w1
      P_Trig( "P_TRIG".ARR[31] )
      S_Coil( "OUTPUT MAPPING DB"."HOOTER RESET" )
   END_RUNG
   // the same network as SCL:
   "IEC_Timer_0_DB_128".TON(IN := "OUTPUT MAPPING DB"."BACK WASH RECOVERY P-801 A" AND NOT "INPUT MAPPING DB"."P-801 A BACK WASH WAST FEED BACK",
                           PT := T#5S);
   "ALARM DB"."BACK WASH RECOVERY P-801 A MPCB_FEEDBACK FAIL" := "IEC_Timer_0_DB_128".Q;
   #_w1 := "IEC_Timer_0_DB_128".Q AND NOT "P_TRIG".ARR[31];   // rising edge
   "P_TRIG".ARR[31] := "IEC_Timer_0_DB_128".Q;
   IF #_w1 THEN "OUTPUT MAPPING DB"."HOOTER RESET" := TRUE; END_IF;
END_REGION

REGION Network 33: BACK WASH RECOVERY P-801 B MPCB_FEEDBACK FAIL
   RUNG wire#powerrail
      Contact( "OUTPUT MAPPING DB"."BACK WASH RECOVERY P-801 B" )
      I_Contact( "INPUT MAPPING DB"."P-801 B BACK WASH WAST FEED BACK" )
      { S7_Templates := "time_type := Time" } "IEC_Timer_0_DB_129".TON(pt := T#5S, et =>)
      wire#w1
      Coil( "ALARM DB"."BACK WASH RECOVERY P-801 B MPCB_FEEDBACK FAIL" )
   END_RUNG
   RUNG wire#w1
      P_Trig( "P_TRIG".ARR[32] )
      S_Coil( "OUTPUT MAPPING DB"."HOOTER RESET" )
   END_RUNG
   // the same network as SCL:
   "IEC_Timer_0_DB_129".TON(IN := "OUTPUT MAPPING DB"."BACK WASH RECOVERY P-801 B" AND NOT "INPUT MAPPING DB"."P-801 B BACK WASH WAST FEED BACK",
                           PT := T#5S);
   "ALARM DB"."BACK WASH RECOVERY P-801 B MPCB_FEEDBACK FAIL" := "IEC_Timer_0_DB_129".Q;
   #_w1 := "IEC_Timer_0_DB_129".Q AND NOT "P_TRIG".ARR[32];   // rising edge
   "P_TRIG".ARR[32] := "IEC_Timer_0_DB_129".Q;
   IF #_w1 THEN "OUTPUT MAPPING DB"."HOOTER RESET" := TRUE; END_IF;
END_REGION

REGION Network 34: UF BACKWASH P-201A_FEEDBACK FAIL
   RUNG wire#powerrail
      Contact( "OUTPUT MAPPING DB"."UF BACK WASH P-201 A" )
      I_Contact( "INPUT MAPPING DB"."P-201 A UF BACK WASH" )
      { S7_Templates := "time_type := Time" } "IEC_Timer_0_DB_130".TON(pt := T#5S, et =>)
      wire#w1
      Coil( "ALARM DB"."UF BACKWASH P-201A_FEEDBACK FAIL" )
   END_RUNG
   RUNG wire#w1
      P_Trig( "P_TRIG".ARR[33] )
      S_Coil( "OUTPUT MAPPING DB"."HOOTER RESET" )
   END_RUNG
   // the same network as SCL:
   "IEC_Timer_0_DB_130".TON(IN := "OUTPUT MAPPING DB"."UF BACK WASH P-201 A" AND NOT "INPUT MAPPING DB"."P-201 A UF BACK WASH",
                           PT := T#5S);
   "ALARM DB"."UF BACKWASH P-201A_FEEDBACK FAIL" := "IEC_Timer_0_DB_130".Q;
   #_w1 := "IEC_Timer_0_DB_130".Q AND NOT "P_TRIG".ARR[33];   // rising edge
   "P_TRIG".ARR[33] := "IEC_Timer_0_DB_130".Q;
   IF #_w1 THEN "OUTPUT MAPPING DB"."HOOTER RESET" := TRUE; END_IF;
END_REGION

REGION Network 35: UF BACKWASH P-201B_FEEDBACK FAIL
   RUNG wire#powerrail
      Contact( "OUTPUT MAPPING DB"."UF BACK WASH  P-201 B" )
      I_Contact( "INPUT MAPPING DB"."P-201 B UF BACK WASH" )
      { S7_Templates := "time_type := Time" } "IEC_Timer_0_DB_131".TON(pt := T#5S, et =>)
      wire#w1
      Coil( "ALARM DB"."UF BACKWASH P-201B_FEEDBACK FAIL" )
   END_RUNG
   RUNG wire#w1
      P_Trig( "P_TRIG".ARR[34] )
      S_Coil( "OUTPUT MAPPING DB"."HOOTER RESET" )
   END_RUNG
   // the same network as SCL:
   "IEC_Timer_0_DB_131".TON(IN := "OUTPUT MAPPING DB"."UF BACK WASH  P-201 B" AND NOT "INPUT MAPPING DB"."P-201 B UF BACK WASH",
                           PT := T#5S);
   "ALARM DB"."UF BACKWASH P-201B_FEEDBACK FAIL" := "IEC_Timer_0_DB_131".Q;
   #_w1 := "IEC_Timer_0_DB_131".Q AND NOT "P_TRIG".ARR[34];   // rising edge
   "P_TRIG".ARR[34] := "IEC_Timer_0_DB_131".Q;
   IF #_w1 THEN "OUTPUT MAPPING DB"."HOOTER RESET" := TRUE; END_IF;
END_REGION

REGION Network 36: MGF INLET VALVE ABFV-101 OPEN COMMOND FAIL
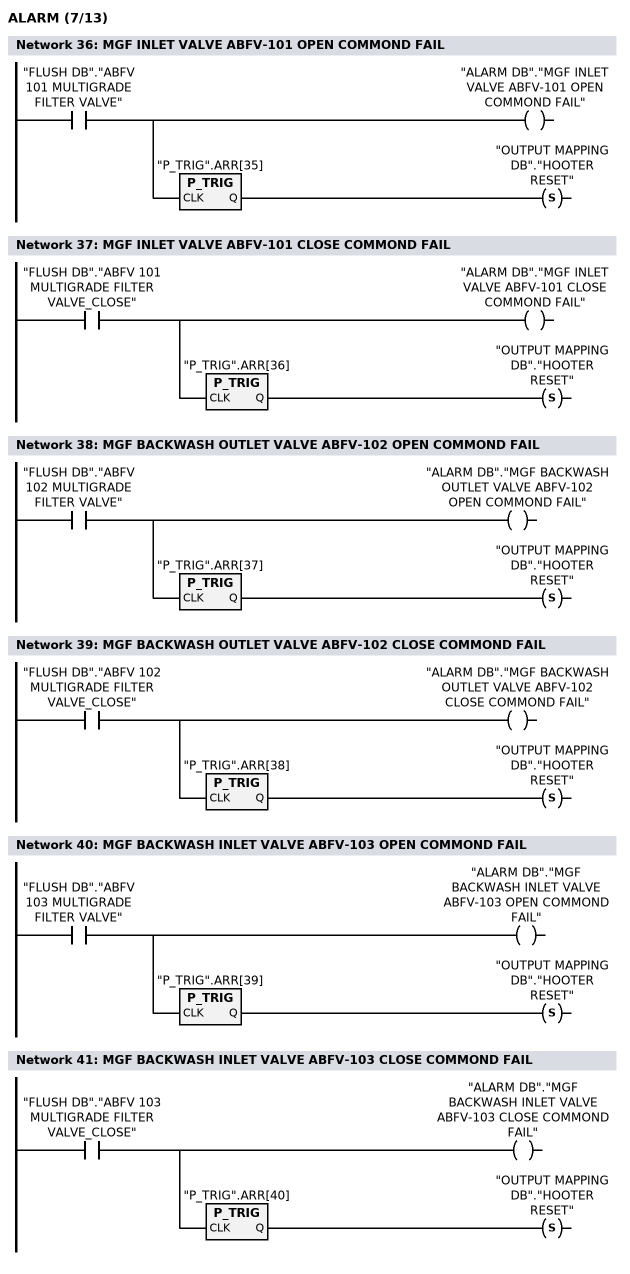
   RUNG wire#powerrail
      Contact( "FLUSH DB"."ABFV 101 MULTIGRADE FILTER VALVE" )
      wire#w1
      Coil( "ALARM DB"."MGF INLET VALVE ABFV-101 OPEN COMMOND FAIL" )
   END_RUNG
   RUNG wire#w1
      P_Trig( "P_TRIG".ARR[35] )
      S_Coil( "OUTPUT MAPPING DB"."HOOTER RESET" )
   END_RUNG
   // the same network as SCL:
   "ALARM DB"."MGF INLET VALVE ABFV-101 OPEN COMMOND FAIL" := "FLUSH DB"."ABFV 101 MULTIGRADE FILTER VALVE";
   #_w1 := "FLUSH DB"."ABFV 101 MULTIGRADE FILTER VALVE" AND NOT "P_TRIG".ARR[35];   // rising edge
   "P_TRIG".ARR[35] := "FLUSH DB"."ABFV 101 MULTIGRADE FILTER VALVE";
   IF #_w1 THEN "OUTPUT MAPPING DB"."HOOTER RESET" := TRUE; END_IF;
END_REGION

REGION Network 37: MGF INLET VALVE ABFV-101 CLOSE COMMOND FAIL
   RUNG wire#powerrail
      Contact( "FLUSH DB"."ABFV 101 MULTIGRADE FILTER VALVE_CLOSE" )
      wire#w1
      Coil( "ALARM DB"."MGF INLET VALVE ABFV-101 CLOSE COMMOND FAIL" )
   END_RUNG
   RUNG wire#w1
      P_Trig( "P_TRIG".ARR[36] )
      S_Coil( "OUTPUT MAPPING DB"."HOOTER RESET" )
   END_RUNG
   // the same network as SCL:
   "ALARM DB"."MGF INLET VALVE ABFV-101 CLOSE COMMOND FAIL" := "FLUSH DB"."ABFV 101 MULTIGRADE FILTER VALVE_CLOSE";
   #_w1 := "FLUSH DB"."ABFV 101 MULTIGRADE FILTER VALVE_CLOSE" AND NOT "P_TRIG".ARR[36];   // rising edge
   "P_TRIG".ARR[36] := "FLUSH DB"."ABFV 101 MULTIGRADE FILTER VALVE_CLOSE";
   IF #_w1 THEN "OUTPUT MAPPING DB"."HOOTER RESET" := TRUE; END_IF;
END_REGION

REGION Network 38: MGF BACKWASH OUTLET VALVE ABFV-102 OPEN COMMOND FAIL
   RUNG wire#powerrail
      Contact( "FLUSH DB"."ABFV 102 MULTIGRADE FILTER VALVE" )
      wire#w1
      Coil( "ALARM DB"."MGF BACKWASH OUTLET VALVE ABFV-102 OPEN COMMOND FAIL" )
   END_RUNG
   RUNG wire#w1
      P_Trig( "P_TRIG".ARR[37] )
      S_Coil( "OUTPUT MAPPING DB"."HOOTER RESET" )
   END_RUNG
   // the same network as SCL:
   "ALARM DB"."MGF BACKWASH OUTLET VALVE ABFV-102 OPEN COMMOND FAIL" := "FLUSH DB"."ABFV 102 MULTIGRADE FILTER VALVE";
   #_w1 := "FLUSH DB"."ABFV 102 MULTIGRADE FILTER VALVE" AND NOT "P_TRIG".ARR[37];   // rising edge
   "P_TRIG".ARR[37] := "FLUSH DB"."ABFV 102 MULTIGRADE FILTER VALVE";
   IF #_w1 THEN "OUTPUT MAPPING DB"."HOOTER RESET" := TRUE; END_IF;
END_REGION

REGION Network 39: MGF BACKWASH OUTLET VALVE ABFV-102 CLOSE COMMOND FAIL
   RUNG wire#powerrail
      Contact( "FLUSH DB"."ABFV 102 MULTIGRADE FILTER VALVE_CLOSE" )
      wire#w1
      Coil( "ALARM DB"."MGF BACKWASH OUTLET VALVE ABFV-102 CLOSE COMMOND FAIL" )
   END_RUNG
   RUNG wire#w1
      P_Trig( "P_TRIG".ARR[38] )
      S_Coil( "OUTPUT MAPPING DB"."HOOTER RESET" )
   END_RUNG
   // the same network as SCL:
   "ALARM DB"."MGF BACKWASH OUTLET VALVE ABFV-102 CLOSE COMMOND FAIL" := "FLUSH DB"."ABFV 102 MULTIGRADE FILTER VALVE_CLOSE";
   #_w1 := "FLUSH DB"."ABFV 102 MULTIGRADE FILTER VALVE_CLOSE" AND NOT "P_TRIG".ARR[38];   // rising edge
   "P_TRIG".ARR[38] := "FLUSH DB"."ABFV 102 MULTIGRADE FILTER VALVE_CLOSE";
   IF #_w1 THEN "OUTPUT MAPPING DB"."HOOTER RESET" := TRUE; END_IF;
END_REGION

REGION Network 40: MGF BACKWASH INLET VALVE ABFV-103 OPEN COMMOND FAIL
   RUNG wire#powerrail
      Contact( "FLUSH DB"."ABFV 103 MULTIGRADE FILTER VALVE" )
      wire#w1
      Coil( "ALARM DB"."MGF BACKWASH INLET VALVE ABFV-103 OPEN COMMOND FAIL" )
   END_RUNG
   RUNG wire#w1
      P_Trig( "P_TRIG".ARR[39] )
      S_Coil( "OUTPUT MAPPING DB"."HOOTER RESET" )
   END_RUNG
   // the same network as SCL:
   "ALARM DB"."MGF BACKWASH INLET VALVE ABFV-103 OPEN COMMOND FAIL" := "FLUSH DB"."ABFV 103 MULTIGRADE FILTER VALVE";
   #_w1 := "FLUSH DB"."ABFV 103 MULTIGRADE FILTER VALVE" AND NOT "P_TRIG".ARR[39];   // rising edge
   "P_TRIG".ARR[39] := "FLUSH DB"."ABFV 103 MULTIGRADE FILTER VALVE";
   IF #_w1 THEN "OUTPUT MAPPING DB"."HOOTER RESET" := TRUE; END_IF;
END_REGION

REGION Network 41: MGF BACKWASH INLET VALVE ABFV-103 CLOSE COMMOND FAIL
   RUNG wire#powerrail
      Contact( "FLUSH DB"."ABFV 103 MULTIGRADE FILTER VALVE_CLOSE" )
      wire#w1
      Coil( "ALARM DB"."MGF BACKWASH INLET VALVE ABFV-103 CLOSE COMMOND FAIL" )
   END_RUNG
   RUNG wire#w1
      P_Trig( "P_TRIG".ARR[40] )
      S_Coil( "OUTPUT MAPPING DB"."HOOTER RESET" )
   END_RUNG
   // the same network as SCL:
   "ALARM DB"."MGF BACKWASH INLET VALVE ABFV-103 CLOSE COMMOND FAIL" := "FLUSH DB"."ABFV 103 MULTIGRADE FILTER VALVE_CLOSE";
   #_w1 := "FLUSH DB"."ABFV 103 MULTIGRADE FILTER VALVE_CLOSE" AND NOT "P_TRIG".ARR[40];   // rising edge
   "P_TRIG".ARR[40] := "FLUSH DB"."ABFV 103 MULTIGRADE FILTER VALVE_CLOSE";
   IF #_w1 THEN "OUTPUT MAPPING DB"."HOOTER RESET" := TRUE; END_IF;
END_REGION

REGION Network 42: MGF OUTLET VALVE ABFV-104 OPEN COMMOND FAIL
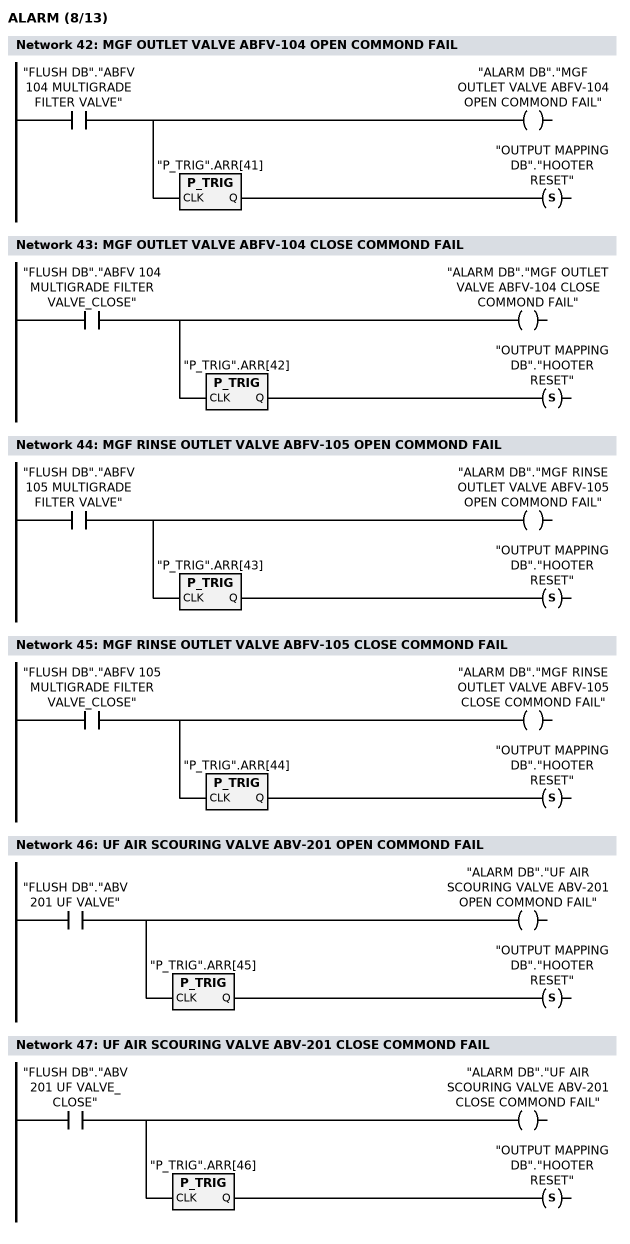
   RUNG wire#powerrail
      Contact( "FLUSH DB"."ABFV 104 MULTIGRADE FILTER VALVE" )
      wire#w1
      Coil( "ALARM DB"."MGF OUTLET VALVE ABFV-104 OPEN COMMOND FAIL" )
   END_RUNG
   RUNG wire#w1
      P_Trig( "P_TRIG".ARR[41] )
      S_Coil( "OUTPUT MAPPING DB"."HOOTER RESET" )
   END_RUNG
   // the same network as SCL:
   "ALARM DB"."MGF OUTLET VALVE ABFV-104 OPEN COMMOND FAIL" := "FLUSH DB"."ABFV 104 MULTIGRADE FILTER VALVE";
   #_w1 := "FLUSH DB"."ABFV 104 MULTIGRADE FILTER VALVE" AND NOT "P_TRIG".ARR[41];   // rising edge
   "P_TRIG".ARR[41] := "FLUSH DB"."ABFV 104 MULTIGRADE FILTER VALVE";
   IF #_w1 THEN "OUTPUT MAPPING DB"."HOOTER RESET" := TRUE; END_IF;
END_REGION

REGION Network 43: MGF OUTLET VALVE ABFV-104 CLOSE COMMOND FAIL
   RUNG wire#powerrail
      Contact( "FLUSH DB"."ABFV 104 MULTIGRADE FILTER VALVE_CLOSE" )
      wire#w1
      Coil( "ALARM DB"."MGF OUTLET VALVE ABFV-104 CLOSE COMMOND FAIL" )
   END_RUNG
   RUNG wire#w1
      P_Trig( "P_TRIG".ARR[42] )
      S_Coil( "OUTPUT MAPPING DB"."HOOTER RESET" )
   END_RUNG
   // the same network as SCL:
   "ALARM DB"."MGF OUTLET VALVE ABFV-104 CLOSE COMMOND FAIL" := "FLUSH DB"."ABFV 104 MULTIGRADE FILTER VALVE_CLOSE";
   #_w1 := "FLUSH DB"."ABFV 104 MULTIGRADE FILTER VALVE_CLOSE" AND NOT "P_TRIG".ARR[42];   // rising edge
   "P_TRIG".ARR[42] := "FLUSH DB"."ABFV 104 MULTIGRADE FILTER VALVE_CLOSE";
   IF #_w1 THEN "OUTPUT MAPPING DB"."HOOTER RESET" := TRUE; END_IF;
END_REGION

REGION Network 44: MGF RINSE OUTLET VALVE ABFV-105 OPEN COMMOND FAIL
   RUNG wire#powerrail
      Contact( "FLUSH DB"."ABFV 105 MULTIGRADE FILTER VALVE" )
      wire#w1
      Coil( "ALARM DB"."MGF RINSE OUTLET VALVE ABFV-105 OPEN COMMOND FAIL" )
   END_RUNG
   RUNG wire#w1
      P_Trig( "P_TRIG".ARR[43] )
      S_Coil( "OUTPUT MAPPING DB"."HOOTER RESET" )
   END_RUNG
   // the same network as SCL:
   "ALARM DB"."MGF RINSE OUTLET VALVE ABFV-105 OPEN COMMOND FAIL" := "FLUSH DB"."ABFV 105 MULTIGRADE FILTER VALVE";
   #_w1 := "FLUSH DB"."ABFV 105 MULTIGRADE FILTER VALVE" AND NOT "P_TRIG".ARR[43];   // rising edge
   "P_TRIG".ARR[43] := "FLUSH DB"."ABFV 105 MULTIGRADE FILTER VALVE";
   IF #_w1 THEN "OUTPUT MAPPING DB"."HOOTER RESET" := TRUE; END_IF;
END_REGION

REGION Network 45: MGF RINSE OUTLET VALVE ABFV-105 CLOSE COMMOND FAIL
   RUNG wire#powerrail
      Contact( "FLUSH DB"."ABFV 105 MULTIGRADE FILTER VALVE_CLOSE" )
      wire#w1
      Coil( "ALARM DB"."MGF RINSE OUTLET VALVE ABFV-105 CLOSE COMMOND FAIL" )
   END_RUNG
   RUNG wire#w1
      P_Trig( "P_TRIG".ARR[44] )
      S_Coil( "OUTPUT MAPPING DB"."HOOTER RESET" )
   END_RUNG
   // the same network as SCL:
   "ALARM DB"."MGF RINSE OUTLET VALVE ABFV-105 CLOSE COMMOND FAIL" := "FLUSH DB"."ABFV 105 MULTIGRADE FILTER VALVE_CLOSE";
   #_w1 := "FLUSH DB"."ABFV 105 MULTIGRADE FILTER VALVE_CLOSE" AND NOT "P_TRIG".ARR[44];   // rising edge
   "P_TRIG".ARR[44] := "FLUSH DB"."ABFV 105 MULTIGRADE FILTER VALVE_CLOSE";
   IF #_w1 THEN "OUTPUT MAPPING DB"."HOOTER RESET" := TRUE; END_IF;
END_REGION

REGION Network 46: UF AIR SCOURING VALVE ABV-201 OPEN COMMOND FAIL
   RUNG wire#powerrail
      Contact( "FLUSH DB"."ABV 201 UF VALVE" )
      wire#w1
      Coil( "ALARM DB"."UF AIR SCOURING VALVE ABV-201 OPEN COMMOND FAIL" )
   END_RUNG
   RUNG wire#w1
      P_Trig( "P_TRIG".ARR[45] )
      S_Coil( "OUTPUT MAPPING DB"."HOOTER RESET" )
   END_RUNG
   // the same network as SCL:
   "ALARM DB"."UF AIR SCOURING VALVE ABV-201 OPEN COMMOND FAIL" := "FLUSH DB"."ABV 201 UF VALVE";
   #_w1 := "FLUSH DB"."ABV 201 UF VALVE" AND NOT "P_TRIG".ARR[45];   // rising edge
   "P_TRIG".ARR[45] := "FLUSH DB"."ABV 201 UF VALVE";
   IF #_w1 THEN "OUTPUT MAPPING DB"."HOOTER RESET" := TRUE; END_IF;
END_REGION

REGION Network 47: UF AIR SCOURING VALVE ABV-201 CLOSE COMMOND FAIL
   RUNG wire#powerrail
      Contact( "FLUSH DB"."ABV 201 UF VALVE_CLOSE" )
      wire#w1
      Coil( "ALARM DB"."UF AIR SCOURING VALVE ABV-201 CLOSE COMMOND FAIL" )
   END_RUNG
   RUNG wire#w1
      P_Trig( "P_TRIG".ARR[46] )
      S_Coil( "OUTPUT MAPPING DB"."HOOTER RESET" )
   END_RUNG
   // the same network as SCL:
   "ALARM DB"."UF AIR SCOURING VALVE ABV-201 CLOSE COMMOND FAIL" := "FLUSH DB"."ABV 201 UF VALVE_CLOSE";
   #_w1 := "FLUSH DB"."ABV 201 UF VALVE_CLOSE" AND NOT "P_TRIG".ARR[46];   // rising edge
   "P_TRIG".ARR[46] := "FLUSH DB"."ABV 201 UF VALVE_CLOSE";
   IF #_w1 THEN "OUTPUT MAPPING DB"."HOOTER RESET" := TRUE; END_IF;
END_REGION

REGION Network 48: UF INLET VALVE ABFV-201 OPEN COMMOND FAIL
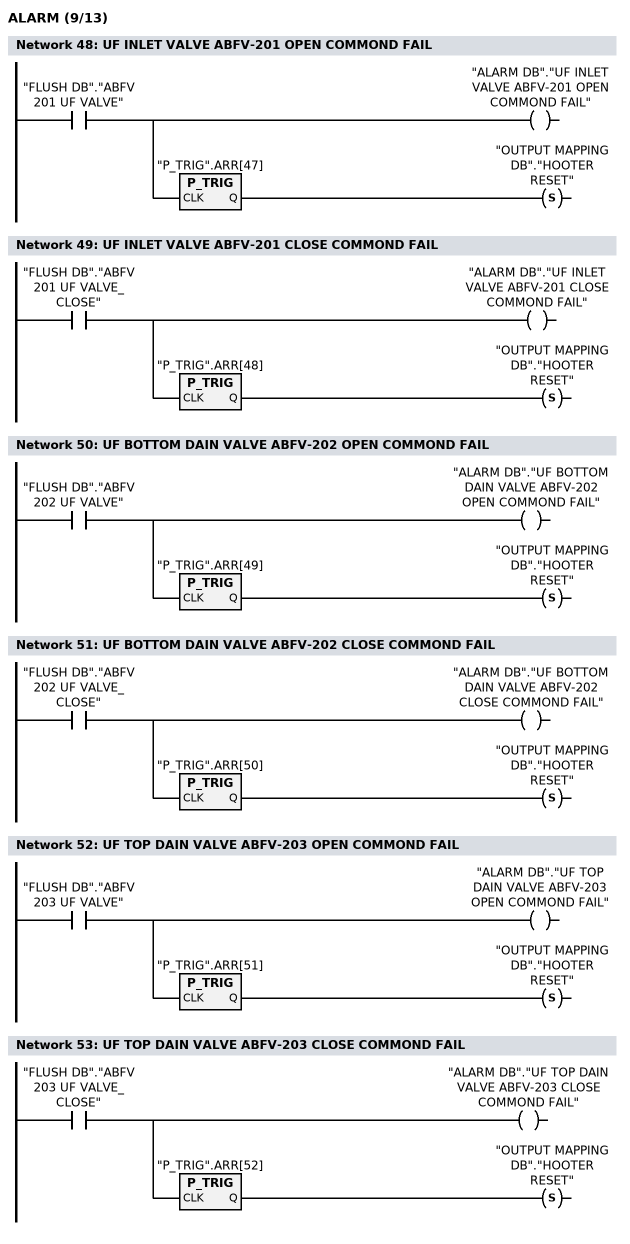
   RUNG wire#powerrail
      Contact( "FLUSH DB"."ABFV 201 UF VALVE" )
      wire#w1
      Coil( "ALARM DB"."UF INLET VALVE ABFV-201 OPEN COMMOND FAIL" )
   END_RUNG
   RUNG wire#w1
      P_Trig( "P_TRIG".ARR[47] )
      S_Coil( "OUTPUT MAPPING DB"."HOOTER RESET" )
   END_RUNG
   // the same network as SCL:
   "ALARM DB"."UF INLET VALVE ABFV-201 OPEN COMMOND FAIL" := "FLUSH DB"."ABFV 201 UF VALVE";
   #_w1 := "FLUSH DB"."ABFV 201 UF VALVE" AND NOT "P_TRIG".ARR[47];   // rising edge
   "P_TRIG".ARR[47] := "FLUSH DB"."ABFV 201 UF VALVE";
   IF #_w1 THEN "OUTPUT MAPPING DB"."HOOTER RESET" := TRUE; END_IF;
END_REGION

REGION Network 49: UF INLET VALVE ABFV-201 CLOSE COMMOND FAIL
   RUNG wire#powerrail
      Contact( "FLUSH DB"."ABFV 201 UF VALVE_CLOSE" )
      wire#w1
      Coil( "ALARM DB"."UF INLET VALVE ABFV-201 CLOSE COMMOND FAIL" )
   END_RUNG
   RUNG wire#w1
      P_Trig( "P_TRIG".ARR[48] )
      S_Coil( "OUTPUT MAPPING DB"."HOOTER RESET" )
   END_RUNG
   // the same network as SCL:
   "ALARM DB"."UF INLET VALVE ABFV-201 CLOSE COMMOND FAIL" := "FLUSH DB"."ABFV 201 UF VALVE_CLOSE";
   #_w1 := "FLUSH DB"."ABFV 201 UF VALVE_CLOSE" AND NOT "P_TRIG".ARR[48];   // rising edge
   "P_TRIG".ARR[48] := "FLUSH DB"."ABFV 201 UF VALVE_CLOSE";
   IF #_w1 THEN "OUTPUT MAPPING DB"."HOOTER RESET" := TRUE; END_IF;
END_REGION

REGION Network 50: UF BOTTOM DAIN VALVE ABFV-202 OPEN COMMOND FAIL
   RUNG wire#powerrail
      Contact( "FLUSH DB"."ABFV 202 UF VALVE" )
      wire#w1
      Coil( "ALARM DB"."UF BOTTOM DAIN VALVE ABFV-202 OPEN COMMOND FAIL" )
   END_RUNG
   RUNG wire#w1
      P_Trig( "P_TRIG".ARR[49] )
      S_Coil( "OUTPUT MAPPING DB"."HOOTER RESET" )
   END_RUNG
   // the same network as SCL:
   "ALARM DB"."UF BOTTOM DAIN VALVE ABFV-202 OPEN COMMOND FAIL" := "FLUSH DB"."ABFV 202 UF VALVE";
   #_w1 := "FLUSH DB"."ABFV 202 UF VALVE" AND NOT "P_TRIG".ARR[49];   // rising edge
   "P_TRIG".ARR[49] := "FLUSH DB"."ABFV 202 UF VALVE";
   IF #_w1 THEN "OUTPUT MAPPING DB"."HOOTER RESET" := TRUE; END_IF;
END_REGION

REGION Network 51: UF BOTTOM DAIN VALVE ABFV-202 CLOSE COMMOND FAIL
   RUNG wire#powerrail
      Contact( "FLUSH DB"."ABFV 202 UF VALVE_CLOSE" )
      wire#w1
      Coil( "ALARM DB"."UF BOTTOM DAIN VALVE ABFV-202 CLOSE COMMOND FAIL" )
   END_RUNG
   RUNG wire#w1
      P_Trig( "P_TRIG".ARR[50] )
      S_Coil( "OUTPUT MAPPING DB"."HOOTER RESET" )
   END_RUNG
   // the same network as SCL:
   "ALARM DB"."UF BOTTOM DAIN VALVE ABFV-202 CLOSE COMMOND FAIL" := "FLUSH DB"."ABFV 202 UF VALVE_CLOSE";
   #_w1 := "FLUSH DB"."ABFV 202 UF VALVE_CLOSE" AND NOT "P_TRIG".ARR[50];   // rising edge
   "P_TRIG".ARR[50] := "FLUSH DB"."ABFV 202 UF VALVE_CLOSE";
   IF #_w1 THEN "OUTPUT MAPPING DB"."HOOTER RESET" := TRUE; END_IF;
END_REGION

REGION Network 52: UF TOP DAIN VALVE ABFV-203 OPEN COMMOND FAIL
   RUNG wire#powerrail
      Contact( "FLUSH DB"."ABFV 203 UF VALVE" )
      wire#w1
      Coil( "ALARM DB"."UF TOP DAIN VALVE ABFV-203 OPEN COMMOND FAIL" )
   END_RUNG
   RUNG wire#w1
      P_Trig( "P_TRIG".ARR[51] )
      S_Coil( "OUTPUT MAPPING DB"."HOOTER RESET" )
   END_RUNG
   // the same network as SCL:
   "ALARM DB"."UF TOP DAIN VALVE ABFV-203 OPEN COMMOND FAIL" := "FLUSH DB"."ABFV 203 UF VALVE";
   #_w1 := "FLUSH DB"."ABFV 203 UF VALVE" AND NOT "P_TRIG".ARR[51];   // rising edge
   "P_TRIG".ARR[51] := "FLUSH DB"."ABFV 203 UF VALVE";
   IF #_w1 THEN "OUTPUT MAPPING DB"."HOOTER RESET" := TRUE; END_IF;
END_REGION

REGION Network 53: UF TOP DAIN VALVE ABFV-203 CLOSE COMMOND FAIL
   RUNG wire#powerrail
      Contact( "FLUSH DB"."ABFV 203 UF VALVE_CLOSE" )
      wire#w1
      Coil( "ALARM DB"."UF TOP DAIN VALVE ABFV-203 CLOSE COMMOND FAIL" )
   END_RUNG
   RUNG wire#w1
      P_Trig( "P_TRIG".ARR[52] )
      S_Coil( "OUTPUT MAPPING DB"."HOOTER RESET" )
   END_RUNG
   // the same network as SCL:
   "ALARM DB"."UF TOP DAIN VALVE ABFV-203 CLOSE COMMOND FAIL" := "FLUSH DB"."ABFV 203 UF VALVE_CLOSE";
   #_w1 := "FLUSH DB"."ABFV 203 UF VALVE_CLOSE" AND NOT "P_TRIG".ARR[52];   // rising edge
   "P_TRIG".ARR[52] := "FLUSH DB"."ABFV 203 UF VALVE_CLOSE";
   IF #_w1 THEN "OUTPUT MAPPING DB"."HOOTER RESET" := TRUE; END_IF;
END_REGION

REGION Network 54: UF BACKWASH INLET VALVE ABFV-204 OPEN COMMOND FAIL
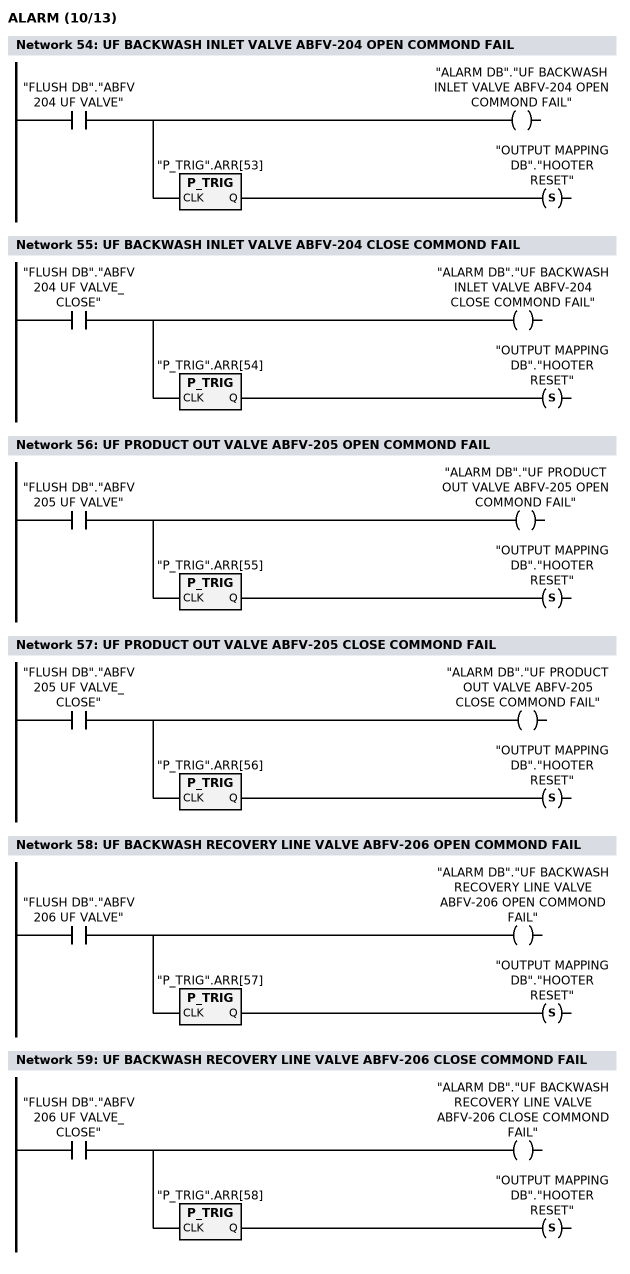
   RUNG wire#powerrail
      Contact( "FLUSH DB"."ABFV 204 UF VALVE" )
      wire#w1
      Coil( "ALARM DB"."UF BACKWASH INLET VALVE ABFV-204 OPEN COMMOND FAIL" )
   END_RUNG
   RUNG wire#w1
      P_Trig( "P_TRIG".ARR[53] )
      S_Coil( "OUTPUT MAPPING DB"."HOOTER RESET" )
   END_RUNG
   // the same network as SCL:
   "ALARM DB"."UF BACKWASH INLET VALVE ABFV-204 OPEN COMMOND FAIL" := "FLUSH DB"."ABFV 204 UF VALVE";
   #_w1 := "FLUSH DB"."ABFV 204 UF VALVE" AND NOT "P_TRIG".ARR[53];   // rising edge
   "P_TRIG".ARR[53] := "FLUSH DB"."ABFV 204 UF VALVE";
   IF #_w1 THEN "OUTPUT MAPPING DB"."HOOTER RESET" := TRUE; END_IF;
END_REGION

REGION Network 55: UF BACKWASH INLET VALVE ABFV-204 CLOSE COMMOND FAIL
   RUNG wire#powerrail
      Contact( "FLUSH DB"."ABFV 204 UF VALVE_CLOSE" )
      wire#w1
      Coil( "ALARM DB"."UF BACKWASH INLET VALVE ABFV-204 CLOSE COMMOND FAIL" )
   END_RUNG
   RUNG wire#w1
      P_Trig( "P_TRIG".ARR[54] )
      S_Coil( "OUTPUT MAPPING DB"."HOOTER RESET" )
   END_RUNG
   // the same network as SCL:
   "ALARM DB"."UF BACKWASH INLET VALVE ABFV-204 CLOSE COMMOND FAIL" := "FLUSH DB"."ABFV 204 UF VALVE_CLOSE";
   #_w1 := "FLUSH DB"."ABFV 204 UF VALVE_CLOSE" AND NOT "P_TRIG".ARR[54];   // rising edge
   "P_TRIG".ARR[54] := "FLUSH DB"."ABFV 204 UF VALVE_CLOSE";
   IF #_w1 THEN "OUTPUT MAPPING DB"."HOOTER RESET" := TRUE; END_IF;
END_REGION

REGION Network 56: UF PRODUCT OUT VALVE ABFV-205 OPEN COMMOND FAIL
   RUNG wire#powerrail
      Contact( "FLUSH DB"."ABFV 205 UF VALVE" )
      wire#w1
      Coil( "ALARM DB"."UF PRODUCT OUT VALVE ABFV-205 OPEN COMMOND FAIL" )
   END_RUNG
   RUNG wire#w1
      P_Trig( "P_TRIG".ARR[55] )
      S_Coil( "OUTPUT MAPPING DB"."HOOTER RESET" )
   END_RUNG
   // the same network as SCL:
   "ALARM DB"."UF PRODUCT OUT VALVE ABFV-205 OPEN COMMOND FAIL" := "FLUSH DB"."ABFV 205 UF VALVE";
   #_w1 := "FLUSH DB"."ABFV 205 UF VALVE" AND NOT "P_TRIG".ARR[55];   // rising edge
   "P_TRIG".ARR[55] := "FLUSH DB"."ABFV 205 UF VALVE";
   IF #_w1 THEN "OUTPUT MAPPING DB"."HOOTER RESET" := TRUE; END_IF;
END_REGION

REGION Network 57: UF PRODUCT OUT VALVE ABFV-205 CLOSE COMMOND FAIL
   RUNG wire#powerrail
      Contact( "FLUSH DB"."ABFV 205 UF VALVE_CLOSE" )
      wire#w1
      Coil( "ALARM DB"."UF PRODUCT OUT VALVE ABFV-205 CLOSE COMMOND FAIL" )
   END_RUNG
   RUNG wire#w1
      P_Trig( "P_TRIG".ARR[56] )
      S_Coil( "OUTPUT MAPPING DB"."HOOTER RESET" )
   END_RUNG
   // the same network as SCL:
   "ALARM DB"."UF PRODUCT OUT VALVE ABFV-205 CLOSE COMMOND FAIL" := "FLUSH DB"."ABFV 205 UF VALVE_CLOSE";
   #_w1 := "FLUSH DB"."ABFV 205 UF VALVE_CLOSE" AND NOT "P_TRIG".ARR[56];   // rising edge
   "P_TRIG".ARR[56] := "FLUSH DB"."ABFV 205 UF VALVE_CLOSE";
   IF #_w1 THEN "OUTPUT MAPPING DB"."HOOTER RESET" := TRUE; END_IF;
END_REGION

REGION Network 58: UF BACKWASH RECOVERY LINE VALVE ABFV-206 OPEN COMMOND FAIL
   RUNG wire#powerrail
      Contact( "FLUSH DB"."ABFV 206 UF VALVE" )
      wire#w1
      Coil( "ALARM DB"."UF BACKWASH RECOVERY LINE VALVE ABFV-206 OPEN COMMOND FAIL" )
   END_RUNG
   RUNG wire#w1
      P_Trig( "P_TRIG".ARR[57] )
      S_Coil( "OUTPUT MAPPING DB"."HOOTER RESET" )
   END_RUNG
   // the same network as SCL:
   "ALARM DB"."UF BACKWASH RECOVERY LINE VALVE ABFV-206 OPEN COMMOND FAIL" := "FLUSH DB"."ABFV 206 UF VALVE";
   #_w1 := "FLUSH DB"."ABFV 206 UF VALVE" AND NOT "P_TRIG".ARR[57];   // rising edge
   "P_TRIG".ARR[57] := "FLUSH DB"."ABFV 206 UF VALVE";
   IF #_w1 THEN "OUTPUT MAPPING DB"."HOOTER RESET" := TRUE; END_IF;
END_REGION

REGION Network 59: UF BACKWASH RECOVERY LINE VALVE ABFV-206 CLOSE COMMOND FAIL
   RUNG wire#powerrail
      Contact( "FLUSH DB"."ABFV 206 UF VALVE_CLOSE" )
      wire#w1
      Coil( "ALARM DB"."UF BACKWASH RECOVERY LINE VALVE ABFV-206 CLOSE COMMOND FAIL" )
   END_RUNG
   RUNG wire#w1
      P_Trig( "P_TRIG".ARR[58] )
      S_Coil( "OUTPUT MAPPING DB"."HOOTER RESET" )
   END_RUNG
   // the same network as SCL:
   "ALARM DB"."UF BACKWASH RECOVERY LINE VALVE ABFV-206 CLOSE COMMOND FAIL" := "FLUSH DB"."ABFV 206 UF VALVE_CLOSE";
   #_w1 := "FLUSH DB"."ABFV 206 UF VALVE_CLOSE" AND NOT "P_TRIG".ARR[58];   // rising edge
   "P_TRIG".ARR[58] := "FLUSH DB"."ABFV 206 UF VALVE_CLOSE";
   IF #_w1 THEN "OUTPUT MAPPING DB"."HOOTER RESET" := TRUE; END_IF;
END_REGION

REGION Network 60: UF BACKWASH DRAIN LINE VALVE ABFV-207 OPEN COMMOND FAIL
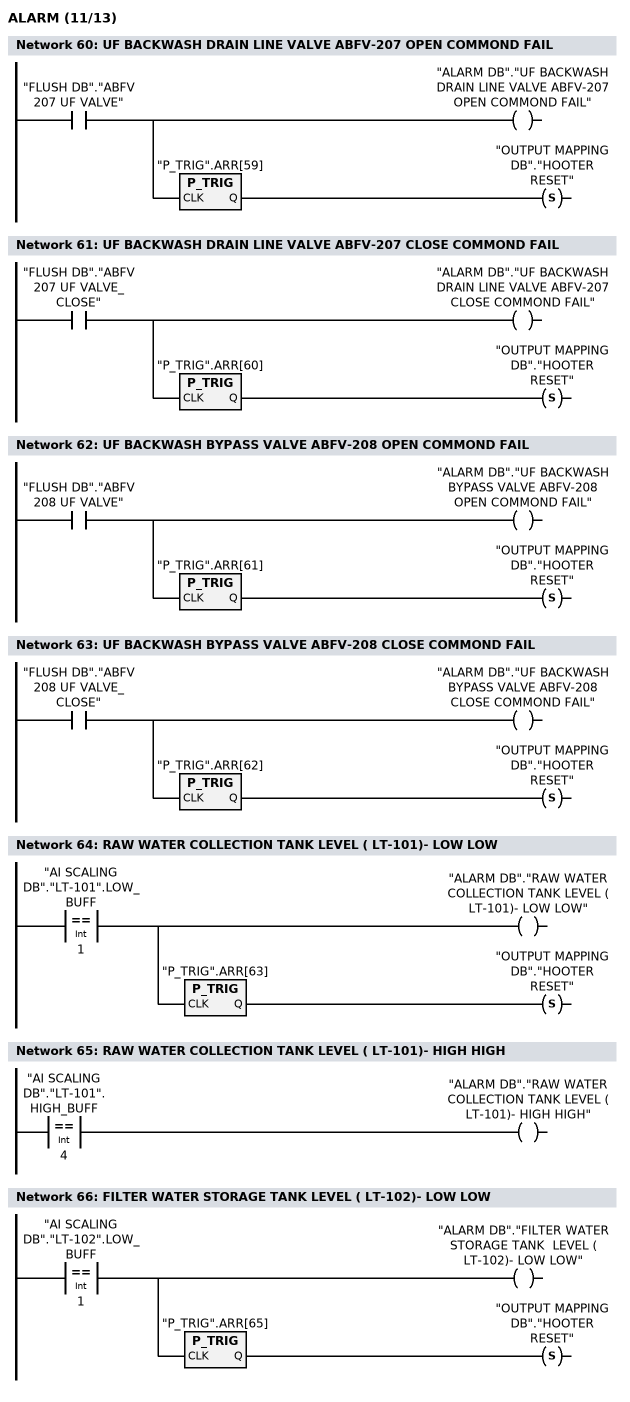
   RUNG wire#powerrail
      Contact( "FLUSH DB"."ABFV 207 UF VALVE" )
      wire#w1
      Coil( "ALARM DB"."UF BACKWASH DRAIN LINE VALVE ABFV-207 OPEN COMMOND FAIL" )
   END_RUNG
   RUNG wire#w1
      P_Trig( "P_TRIG".ARR[59] )
      S_Coil( "OUTPUT MAPPING DB"."HOOTER RESET" )
   END_RUNG
   // the same network as SCL:
   "ALARM DB"."UF BACKWASH DRAIN LINE VALVE ABFV-207 OPEN COMMOND FAIL" := "FLUSH DB"."ABFV 207 UF VALVE";
   #_w1 := "FLUSH DB"."ABFV 207 UF VALVE" AND NOT "P_TRIG".ARR[59];   // rising edge
   "P_TRIG".ARR[59] := "FLUSH DB"."ABFV 207 UF VALVE";
   IF #_w1 THEN "OUTPUT MAPPING DB"."HOOTER RESET" := TRUE; END_IF;
END_REGION

REGION Network 61: UF BACKWASH DRAIN LINE VALVE ABFV-207 CLOSE COMMOND FAIL
   RUNG wire#powerrail
      Contact( "FLUSH DB"."ABFV 207 UF VALVE_CLOSE" )
      wire#w1
      Coil( "ALARM DB"."UF BACKWASH DRAIN LINE VALVE ABFV-207 CLOSE COMMOND FAIL" )
   END_RUNG
   RUNG wire#w1
      P_Trig( "P_TRIG".ARR[60] )
      S_Coil( "OUTPUT MAPPING DB"."HOOTER RESET" )
   END_RUNG
   // the same network as SCL:
   "ALARM DB"."UF BACKWASH DRAIN LINE VALVE ABFV-207 CLOSE COMMOND FAIL" := "FLUSH DB"."ABFV 207 UF VALVE_CLOSE";
   #_w1 := "FLUSH DB"."ABFV 207 UF VALVE_CLOSE" AND NOT "P_TRIG".ARR[60];   // rising edge
   "P_TRIG".ARR[60] := "FLUSH DB"."ABFV 207 UF VALVE_CLOSE";
   IF #_w1 THEN "OUTPUT MAPPING DB"."HOOTER RESET" := TRUE; END_IF;
END_REGION

REGION Network 62: UF BACKWASH BYPASS VALVE ABFV-208 OPEN COMMOND FAIL
   RUNG wire#powerrail
      Contact( "FLUSH DB"."ABFV 208 UF VALVE" )
      wire#w1
      Coil( "ALARM DB"."UF BACKWASH BYPASS VALVE ABFV-208 OPEN COMMOND FAIL" )
   END_RUNG
   RUNG wire#w1
      P_Trig( "P_TRIG".ARR[61] )
      S_Coil( "OUTPUT MAPPING DB"."HOOTER RESET" )
   END_RUNG
   // the same network as SCL:
   "ALARM DB"."UF BACKWASH BYPASS VALVE ABFV-208 OPEN COMMOND FAIL" := "FLUSH DB"."ABFV 208 UF VALVE";
   #_w1 := "FLUSH DB"."ABFV 208 UF VALVE" AND NOT "P_TRIG".ARR[61];   // rising edge
   "P_TRIG".ARR[61] := "FLUSH DB"."ABFV 208 UF VALVE";
   IF #_w1 THEN "OUTPUT MAPPING DB"."HOOTER RESET" := TRUE; END_IF;
END_REGION

REGION Network 63: UF BACKWASH BYPASS VALVE ABFV-208 CLOSE COMMOND FAIL
   RUNG wire#powerrail
      Contact( "FLUSH DB"."ABFV 208 UF VALVE_CLOSE" )
      wire#w1
      Coil( "ALARM DB"."UF BACKWASH BYPASS VALVE ABFV-208 CLOSE COMMOND FAIL" )
   END_RUNG
   RUNG wire#w1
      P_Trig( "P_TRIG".ARR[62] )
      S_Coil( "OUTPUT MAPPING DB"."HOOTER RESET" )
   END_RUNG
   // the same network as SCL:
   "ALARM DB"."UF BACKWASH BYPASS VALVE ABFV-208 CLOSE COMMOND FAIL" := "FLUSH DB"."ABFV 208 UF VALVE_CLOSE";
   #_w1 := "FLUSH DB"."ABFV 208 UF VALVE_CLOSE" AND NOT "P_TRIG".ARR[62];   // rising edge
   "P_TRIG".ARR[62] := "FLUSH DB"."ABFV 208 UF VALVE_CLOSE";
   IF #_w1 THEN "OUTPUT MAPPING DB"."HOOTER RESET" := TRUE; END_IF;
END_REGION

REGION Network 64: RAW WATER COLLECTION TANK LEVEL ( LT-101)- LOW LOW
   RUNG wire#powerrail
      { S7_Templates := "SrcType := Int" } EQ_Contact(in1 := "AI SCALING DB"."LT-101".LOW_BUFF, in2 := 1)
      wire#w1
      Coil( "ALARM DB"."RAW WATER COLLECTION TANK LEVEL ( LT-101)- LOW LOW" )
   END_RUNG
   RUNG wire#w1
      P_Trig( "P_TRIG".ARR[63] )
      S_Coil( "OUTPUT MAPPING DB"."HOOTER RESET" )
   END_RUNG
   // the same network as SCL:
   "ALARM DB"."RAW WATER COLLECTION TANK LEVEL ( LT-101)- LOW LOW" := "AI SCALING DB"."LT-101".LOW_BUFF = 1;
   #_w1 := "ALARM DB"."RAW WATER COLLECTION TANK LEVEL ( LT-101)- LOW LOW" AND NOT "P_TRIG".ARR[63];   // rising edge
   "P_TRIG".ARR[63] := "ALARM DB"."RAW WATER COLLECTION TANK LEVEL ( LT-101)- LOW LOW";
   IF #_w1 THEN "OUTPUT MAPPING DB"."HOOTER RESET" := TRUE; END_IF;
END_REGION

REGION Network 65: RAW WATER COLLECTION TANK LEVEL ( LT-101)- HIGH HIGH
   RUNG wire#powerrail
      { S7_Templates := "SrcType := Int" } EQ_Contact(in1 := "AI SCALING DB"."LT-101".HIGH_BUFF, in2 := 4)
      Coil( "ALARM DB"."RAW WATER COLLECTION TANK LEVEL ( LT-101)- HIGH HIGH" )
   END_RUNG
   // the same network as SCL:
   "ALARM DB"."RAW WATER COLLECTION TANK LEVEL ( LT-101)- HIGH HIGH" := "AI SCALING DB"."LT-101".HIGH_BUFF = 4;
END_REGION

REGION Network 66: FILTER WATER STORAGE TANK LEVEL ( LT-102)- LOW LOW
   RUNG wire#powerrail
      { S7_Templates := "SrcType := Int" } EQ_Contact(in1 := "AI SCALING DB"."LT-102".LOW_BUFF, in2 := 1)
      wire#w1
      Coil( "ALARM DB"."FILTER WATER STORAGE TANK  LEVEL ( LT-102)- LOW LOW" )
   END_RUNG
   RUNG wire#w1
      P_Trig( "P_TRIG".ARR[65] )
      S_Coil( "OUTPUT MAPPING DB"."HOOTER RESET" )
   END_RUNG
   // the same network as SCL:
   "ALARM DB"."FILTER WATER STORAGE TANK  LEVEL ( LT-102)- LOW LOW" := "AI SCALING DB"."LT-102".LOW_BUFF = 1;
   #_w1 := "ALARM DB"."FILTER WATER STORAGE TANK  LEVEL ( LT-102)- LOW LOW" AND NOT "P_TRIG".ARR[65];   // rising edge
   "P_TRIG".ARR[65] := "ALARM DB"."FILTER WATER STORAGE TANK  LEVEL ( LT-102)- LOW LOW";
   IF #_w1 THEN "OUTPUT MAPPING DB"."HOOTER RESET" := TRUE; END_IF;
END_REGION

REGION Network 67: FILTER WATER STORAGE TANK LEVEL ( LT-102)- HIGH HIGH
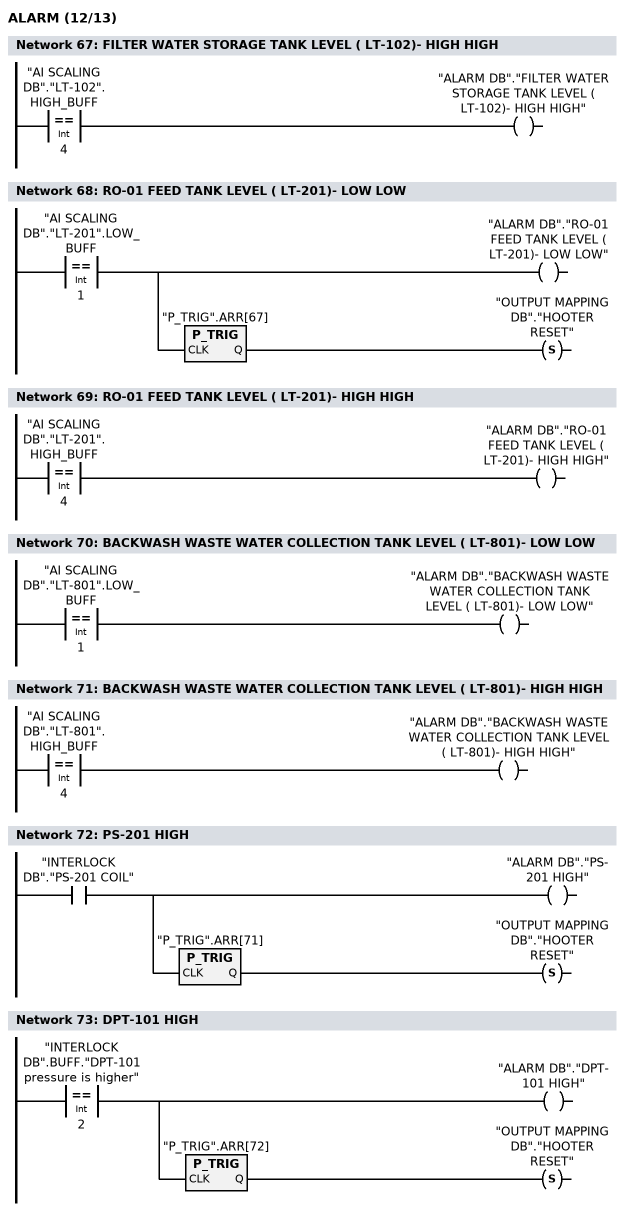
   RUNG wire#powerrail
      { S7_Templates := "SrcType := Int" } EQ_Contact(in1 := "AI SCALING DB"."LT-102".HIGH_BUFF, in2 := 4)
      Coil( "ALARM DB"."FILTER WATER STORAGE TANK LEVEL ( LT-102)- HIGH HIGH" )
   END_RUNG
   // the same network as SCL:
   "ALARM DB"."FILTER WATER STORAGE TANK LEVEL ( LT-102)- HIGH HIGH" := "AI SCALING DB"."LT-102".HIGH_BUFF = 4;
END_REGION

REGION Network 68: RO-01 FEED TANK LEVEL ( LT-201)- LOW LOW
   RUNG wire#powerrail
      { S7_Templates := "SrcType := Int" } EQ_Contact(in1 := "AI SCALING DB"."LT-201".LOW_BUFF, in2 := 1)
      wire#w1
      Coil( "ALARM DB"."RO-01 FEED TANK LEVEL ( LT-201)- LOW LOW" )
   END_RUNG
   RUNG wire#w1
      P_Trig( "P_TRIG".ARR[67] )
      S_Coil( "OUTPUT MAPPING DB"."HOOTER RESET" )
   END_RUNG
   // the same network as SCL:
   "ALARM DB"."RO-01 FEED TANK LEVEL ( LT-201)- LOW LOW" := "AI SCALING DB"."LT-201".LOW_BUFF = 1;
   #_w1 := "ALARM DB"."RO-01 FEED TANK LEVEL ( LT-201)- LOW LOW" AND NOT "P_TRIG".ARR[67];   // rising edge
   "P_TRIG".ARR[67] := "ALARM DB"."RO-01 FEED TANK LEVEL ( LT-201)- LOW LOW";
   IF #_w1 THEN "OUTPUT MAPPING DB"."HOOTER RESET" := TRUE; END_IF;
END_REGION

REGION Network 69: RO-01 FEED TANK LEVEL ( LT-201)- HIGH HIGH
   RUNG wire#powerrail
      { S7_Templates := "SrcType := Int" } EQ_Contact(in1 := "AI SCALING DB"."LT-201".HIGH_BUFF, in2 := 4)
      Coil( "ALARM DB"."RO-01 FEED TANK LEVEL ( LT-201)- HIGH HIGH" )
   END_RUNG
   // the same network as SCL:
   "ALARM DB"."RO-01 FEED TANK LEVEL ( LT-201)- HIGH HIGH" := "AI SCALING DB"."LT-201".HIGH_BUFF = 4;
END_REGION

REGION Network 70: BACKWASH WASTE WATER COLLECTION TANK LEVEL ( LT-801)- LOW LOW
   RUNG wire#powerrail
      { S7_Templates := "SrcType := Int" } EQ_Contact(in1 := "AI SCALING DB"."LT-801".LOW_BUFF, in2 := 1)
      Coil( "ALARM DB"."BACKWASH WASTE WATER COLLECTION TANK  LEVEL ( LT-801)- LOW LOW" )
   END_RUNG
   // the same network as SCL:
   "ALARM DB"."BACKWASH WASTE WATER COLLECTION TANK  LEVEL ( LT-801)- LOW LOW" := "AI SCALING DB"."LT-801".LOW_BUFF = 1;
END_REGION

REGION Network 71: BACKWASH WASTE WATER COLLECTION TANK LEVEL ( LT-801)- HIGH HIGH
   RUNG wire#powerrail
      { S7_Templates := "SrcType := Int" } EQ_Contact(in1 := "AI SCALING DB"."LT-801".HIGH_BUFF, in2 := 4)
      Coil( "ALARM DB"."BACKWASH WASTE WATER COLLECTION TANK LEVEL ( LT-801)- HIGH HIGH" )
   END_RUNG
   // the same network as SCL:
   "ALARM DB"."BACKWASH WASTE WATER COLLECTION TANK LEVEL ( LT-801)- HIGH HIGH" := "AI SCALING DB"."LT-801".HIGH_BUFF = 4;
END_REGION

REGION Network 72: PS-201 HIGH
   RUNG wire#powerrail
      Contact( "INTERLOCK DB"."PS-201 COIL" )
      wire#w1
      Coil( "ALARM DB"."PS-201 HIGH" )
   END_RUNG
   RUNG wire#w1
      P_Trig( "P_TRIG".ARR[71] )
      S_Coil( "OUTPUT MAPPING DB"."HOOTER RESET" )
   END_RUNG
   // the same network as SCL:
   "ALARM DB"."PS-201 HIGH" := "INTERLOCK DB"."PS-201 COIL";
   #_w1 := "INTERLOCK DB"."PS-201 COIL" AND NOT "P_TRIG".ARR[71];   // rising edge
   "P_TRIG".ARR[71] := "INTERLOCK DB"."PS-201 COIL";
   IF #_w1 THEN "OUTPUT MAPPING DB"."HOOTER RESET" := TRUE; END_IF;
END_REGION

REGION Network 73: DPT-101 HIGH
   RUNG wire#powerrail
      { S7_Templates := "SrcType := Int" } EQ_Contact(in1 := "INTERLOCK DB".BUFF."DPT-101 pressure is higher", in2 := 2)
      wire#w1
      Coil( "ALARM DB"."DPT-101 HIGH" )
   END_RUNG
   RUNG wire#w1
      P_Trig( "P_TRIG".ARR[72] )
      S_Coil( "OUTPUT MAPPING DB"."HOOTER RESET" )
   END_RUNG
   // the same network as SCL:
   "ALARM DB"."DPT-101 HIGH" := "INTERLOCK DB".BUFF."DPT-101 pressure is higher" = 2;
   #_w1 := "ALARM DB"."DPT-101 HIGH" AND NOT "P_TRIG".ARR[72];   // rising edge
   "P_TRIG".ARR[72] := "ALARM DB"."DPT-101 HIGH";
   IF #_w1 THEN "OUTPUT MAPPING DB"."HOOTER RESET" := TRUE; END_IF;
END_REGION

REGION Network 74: DPT-201 HIGH
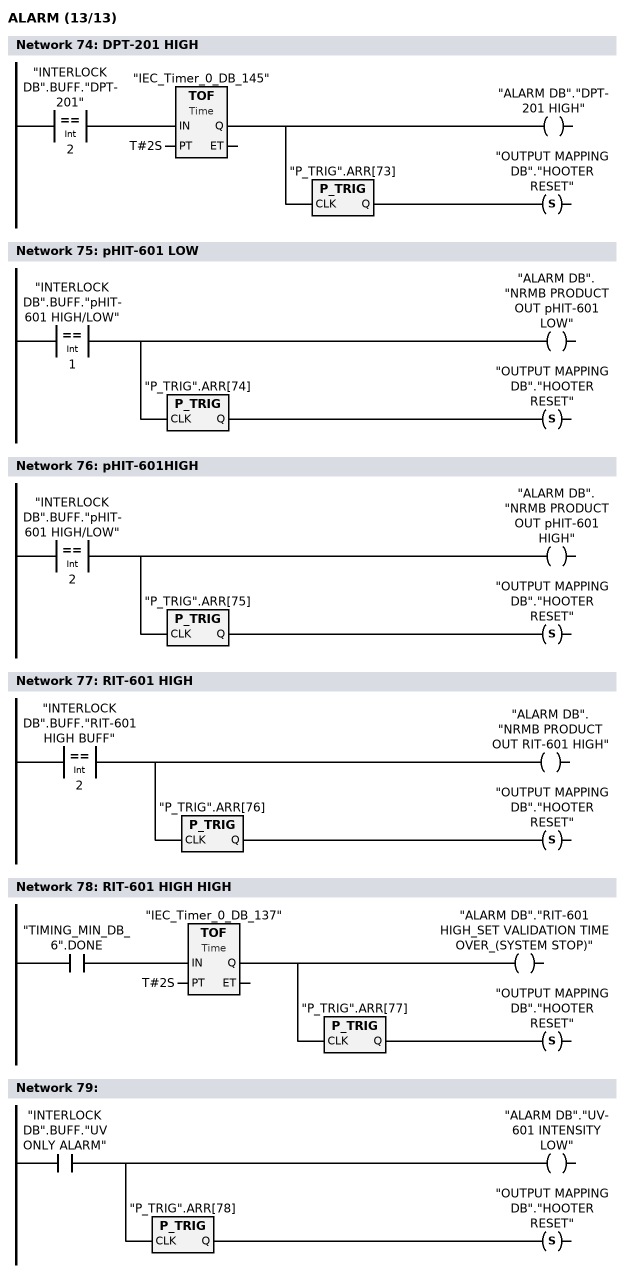
   RUNG wire#powerrail
      { S7_Templates := "SrcType := Int" } EQ_Contact(in1 := "INTERLOCK DB".BUFF."DPT-201", in2 := 2)
      { S7_Templates := "time_type := Time" } "IEC_Timer_0_DB_145".TOF(pt := T#2S, et =>)
      wire#w1
      Coil( "ALARM DB"."DPT-201 HIGH" )
   END_RUNG
   RUNG wire#w1
      P_Trig( "P_TRIG".ARR[73] )
      S_Coil( "OUTPUT MAPPING DB"."HOOTER RESET" )
   END_RUNG
   // the same network as SCL:
   "IEC_Timer_0_DB_145".TOF(IN := "INTERLOCK DB".BUFF."DPT-201" = 2, PT := T#2S);
   "ALARM DB"."DPT-201 HIGH" := "IEC_Timer_0_DB_145".Q;
   #_w1 := "IEC_Timer_0_DB_145".Q AND NOT "P_TRIG".ARR[73];   // rising edge
   "P_TRIG".ARR[73] := "IEC_Timer_0_DB_145".Q;
   IF #_w1 THEN "OUTPUT MAPPING DB"."HOOTER RESET" := TRUE; END_IF;
END_REGION

REGION Network 75: pHIT-601 LOW
   RUNG wire#powerrail
      { S7_Templates := "SrcType := Int" } EQ_Contact(in1 := "INTERLOCK DB".BUFF."pHIT-601 HIGH/LOW", in2 := 1)
      wire#w1
      Coil( "ALARM DB"."NRMB PRODUCT OUT pHIT-601 LOW" )
   END_RUNG
   RUNG wire#w1
      P_Trig( "P_TRIG".ARR[74] )
      S_Coil( "OUTPUT MAPPING DB"."HOOTER RESET" )
   END_RUNG
   // the same network as SCL:
   "ALARM DB"."NRMB PRODUCT OUT pHIT-601 LOW" := "INTERLOCK DB".BUFF."pHIT-601 HIGH/LOW" = 1;
   #_w1 := "ALARM DB"."NRMB PRODUCT OUT pHIT-601 LOW" AND NOT "P_TRIG".ARR[74];   // rising edge
   "P_TRIG".ARR[74] := "ALARM DB"."NRMB PRODUCT OUT pHIT-601 LOW";
   IF #_w1 THEN "OUTPUT MAPPING DB"."HOOTER RESET" := TRUE; END_IF;
END_REGION

REGION Network 76: pHIT-601HIGH
   RUNG wire#powerrail
      { S7_Templates := "SrcType := Int" } EQ_Contact(in1 := "INTERLOCK DB".BUFF."pHIT-601 HIGH/LOW", in2 := 2)
      wire#w1
      Coil( "ALARM DB"."NRMB PRODUCT OUT pHIT-601 HIGH" )
   END_RUNG
   RUNG wire#w1
      P_Trig( "P_TRIG".ARR[75] )
      S_Coil( "OUTPUT MAPPING DB"."HOOTER RESET" )
   END_RUNG
   // the same network as SCL:
   "ALARM DB"."NRMB PRODUCT OUT pHIT-601 HIGH" := "INTERLOCK DB".BUFF."pHIT-601 HIGH/LOW" = 2;
   #_w1 := "ALARM DB"."NRMB PRODUCT OUT pHIT-601 HIGH" AND NOT "P_TRIG".ARR[75];   // rising edge
   "P_TRIG".ARR[75] := "ALARM DB"."NRMB PRODUCT OUT pHIT-601 HIGH";
   IF #_w1 THEN "OUTPUT MAPPING DB"."HOOTER RESET" := TRUE; END_IF;
END_REGION

REGION Network 77: RIT-601 HIGH
   RUNG wire#powerrail
      { S7_Templates := "SrcType := Int" } EQ_Contact(in1 := "INTERLOCK DB".BUFF."RIT-601 HIGH BUFF", in2 := 2)
      wire#w1
      Coil( "ALARM DB"."NRMB PRODUCT OUT RIT-601 HIGH" )
   END_RUNG
   RUNG wire#w1
      P_Trig( "P_TRIG".ARR[76] )
      S_Coil( "OUTPUT MAPPING DB"."HOOTER RESET" )
   END_RUNG
   // the same network as SCL:
   "ALARM DB"."NRMB PRODUCT OUT RIT-601 HIGH" := "INTERLOCK DB".BUFF."RIT-601 HIGH BUFF" = 2;
   #_w1 := "ALARM DB"."NRMB PRODUCT OUT RIT-601 HIGH" AND NOT "P_TRIG".ARR[76];   // rising edge
   "P_TRIG".ARR[76] := "ALARM DB"."NRMB PRODUCT OUT RIT-601 HIGH";
   IF #_w1 THEN "OUTPUT MAPPING DB"."HOOTER RESET" := TRUE; END_IF;
END_REGION

REGION Network 78: RIT-601 HIGH HIGH
   RUNG wire#powerrail
      Contact( "TIMING_MIN_DB_6".DONE )
      { S7_Templates := "time_type := Time" } "IEC_Timer_0_DB_137".TOF(pt := T#2S, et =>)
      wire#w1
      Coil( "ALARM DB"."RIT-601 HIGH_SET VALIDATION TIME OVER_(SYSTEM STOP)" )
   END_RUNG
   RUNG wire#w1
      P_Trig( "P_TRIG".ARR[77] )
      S_Coil( "OUTPUT MAPPING DB"."HOOTER RESET" )
   END_RUNG
   // the same network as SCL:
   "IEC_Timer_0_DB_137".TOF(IN := "TIMING_MIN_DB_6".DONE, PT := T#2S);
   "ALARM DB"."RIT-601 HIGH_SET VALIDATION TIME OVER_(SYSTEM STOP)" := "IEC_Timer_0_DB_137".Q;
   #_w1 := "IEC_Timer_0_DB_137".Q AND NOT "P_TRIG".ARR[77];   // rising edge
   "P_TRIG".ARR[77] := "IEC_Timer_0_DB_137".Q;
   IF #_w1 THEN "OUTPUT MAPPING DB"."HOOTER RESET" := TRUE; END_IF;
END_REGION

REGION Network 79
   RUNG wire#powerrail
      Contact( "INTERLOCK DB".BUFF."UV ONLY ALARM" )
      wire#w1
      Coil( "ALARM DB"."UV-601 INTENSITY LOW" )
   END_RUNG
   RUNG wire#w1
      P_Trig( "P_TRIG".ARR[78] )
      S_Coil( "OUTPUT MAPPING DB"."HOOTER RESET" )
   END_RUNG
   // the same network as SCL:
   "ALARM DB"."UV-601 INTENSITY LOW" := "INTERLOCK DB".BUFF."UV ONLY ALARM";
   #_w1 := "INTERLOCK DB".BUFF."UV ONLY ALARM" AND NOT "P_TRIG".ARR[78];   // rising edge
   "P_TRIG".ARR[78] := "INTERLOCK DB".BUFF."UV ONLY ALARM";
   IF #_w1 THEN "OUTPUT MAPPING DB"."HOOTER RESET" := TRUE; END_IF;
END_REGION
END_FUNCTION
